// TwinCAT 3 PLC project PLC_ST40
// ProgramVersion: 3.1.4023.0
// libraries:
//   Tc2_DataExchange, * (Beckhoff Automation GmbH)
//   Tc2_IoFunctions, * (Beckhoff Automation GmbH)
//   Tc2_MC2, * (Beckhoff Automation GmbH)
//   Tc2_MC2_Drive, * (Beckhoff Automation GmbH)
//   Tc2_Standard, * (Beckhoff Automation GmbH)
//   Tc2_System, * (Beckhoff Automation GmbH)
//   Tc2_TcpIp, * (Beckhoff Automation GmbH)
//   Tc2_Utilities, * (Beckhoff Automation GmbH)
//   Tc3_EventLogger, * (Beckhoff Automation GmbH)
//   Tc3_Harman_MES_Interface, * (Harman)
//   Tc3_Module, * (Beckhoff Automation GmbH)
//   Tc3_Utilities_Extension, * (Harman)
// project tree:
//   DUTs/Camera/ ST_Camera_IN.TcDUT (not stored), ST_Camera_OUT.TcDUT (not stored)
//   DUTs/ENUMERATORs/ ENUM_AXIS_NAME.TcDUT, ENUM_CHANNEL.TcDUT, ENUM_PROCESS.TcDUT, ENUM_PROCESS_RESULT.TcDUT, ENUM_PROCESS_STATE.TcDUT, ENUM_SCREW_FEEDER.TcDUT, ENUM_SLOT.TcDUT, ENUM_SLOT_STATE.TcDUT, ENUM_SLOT_TYPE.TcDUT, ENUM_STATION.TcDUT
//   DUTs/ E_ADS_Cmd.TcTLEO (not stored), ST_CamSeq.TcDUT, ST_Coordinates_XYZ.TcDUT, ST_P1MesData.TcDUT, ST_PalletData.TcDUT, ST_PosData.TcDUT, ST_ProductData.TcDUT (not stored)
//   DUTs/Kuka/ ST_KRC_Control.TcDUT, ST_KRC_Status.TcDUT (not stored), U_KRC_Input.TcDUT, U_KRC_Output.TcDUT (not stored)
//   DUTs/NewFolder1/ ST_MOVE.TcDUT, ST_SCREWING.TcDUT, ST_SCR_RECIPE.TcDUT, ST_Vision.TcDUT
//   DUTs/PERSISTENT_STs/ ST_CONFIG.TcDUT
//   DUTs/STRUCTUREs/NewFolder1/ ST_MOVE_1.TcDUT, ST_SCREWING_1.TcDUT, ST_SCR_RECIPE_1.TcDUT
//   DUTs/STRUCTUREs/PROCESS_PARAM/MACHINE/ ST_P_BARCODE_READ.TcDUT, ST_P_CAMERA.TcDUT, ST_P_CHECK_INPUT.TcDUT, ST_P_MOVE.TcDUT, ST_P_RELEASE_PARTS.TcDUT, ST_P_RESET.TcDUT, ST_P_SCREWING.TcDUT, ST_P_SET.TcDUT, ST_P_SET_RECIPE.TcDUT, ST_P_SET_RECIPE_COND.TcDUT, ST_P_TAKE_SCREW.TcDUT, ST_P_WAIT.TcDUT, ST_P_WAIT_UNTIL.TcDUT
//   DUTs/STRUCTUREs/PROCESS_PARAM/MES/ ST_P_ASSY_ELEMENT.TcDUT, ST_P_CHECK_TIMECONTROL.TcDUT, ST_P_COMPLETE_ASSY.TcDUT, ST_P_COMPLETE_OP.TcDUT, ST_P_GET_CHILD.TcDUT, ST_P_GET_OP_STATE.TcDUT, ST_P_GET_PARENT.TcDUT, ST_P_GET_RECIPE.TcDUT, ST_P_RELEASE_MRT.TcDUT, ST_P_SAVE_MESDAT.TcDUT, ST_P_START_ASSY.TcDUT, ST_P_START_OP.TcDUT, ST_P_STOP_TIMECONTROL.TcDUT
//   DUTs/STRUCTUREs/ ST_COORDINATE.TcDUT, ST_DEPTH_DATA_DUT.TcDUT, ST_PARAMETER_COLLECTION.TcDUT, ST_PROCESS.TcDUT, ST_RECIPE.TcDUT, ST_SLOT_VISUALISATION.TcDUT
//   GVLs/ GVL_Constant.TcGVL, GVL_IO.TcGVL, GVL_Main.TcGVL, GVL_Persistenet.TcGVL, GVL_Recipe.TcGVL, GVL_Safety.TcGVL
//   / PlcTask.TcTTO
//   POUs/ Blink.TcPOU, Conveyor.TcPOU, Diag.TcPOU, Lift.TcPOU (not stored), MAIN.TcPOU, MesTest.TcPOU, P1_Camera.TcPOU, P2_Robot.TcPOU
//   POUs/FBs/ FB_ADSHandler.TcPOU (not stored), FB_BISL.TcPOU, FB_BISM.TcPOU, FB_Bistabil.TcPOU (not stored), FB_Conveyor.TcPOU, FB_Door.TcPOU, FB_FullCycleTime.TcPOU, FB_GenPulse.TcPOU (not stored), FB_KRC4.TcPOU, FB_Motor.TcPOU (not stored), FB_ReceipeList.TcPOU, FB_Stopper.TcPOU (not stored), FB_Stopper2.TcPOU (not stored), FB_TcEvent.TcPOU (not stored), FB_UpsC69xx.TcPOU, FB_UserLed.TcPOU, FB_WorkLight.TcPOU
//   POUs/FBs/FB_Camera/ FB_Kamino.TcPOU (not stored)
//   POUs/FBs/SmartLight/DUT/ E_BlinkFrequency.TcDUT (not stored), E_BuzzerType.TcDUT (not stored), E_Color.TcDUT, E_Mode.TcDUT (not stored)
//   POUs/FBs/SmartLight/ FB_SmartLight.TcPOU (not stored)
// real-time tasks:
//   TASK PlcTask: cycle T#10ms, priority 20, ADS port 350
// I/O:
//   DEVICE Device 4 (EtherCAT), AmsNetId 192.168.102.141.5.1
//     Term 1 (EK1100) [EK1100 EtherCAT Coupler (2A E-Bus)]
//       Term 2 (EL1918) [EL1918, 8Ch. Safety Input 24V, TwinSAFE]
//         modules: Module 2 (FSLOGIC)
//       Term 3 (EL2904) [EL2904, 4 Ch. Safety Output 24V, 0.5A, TwinSAFE]
//         modules: Module 1 (FSOES), Module 2 (DO)
//       Term 4 (EL2904) [EL2904, 4 Ch. Safety Output 24V, 0.5A, TwinSAFE]
//         modules: Module 1 (FSOES), Module 2 (DO)
//       Term 5 (EL1809) [EL1809 16Ch. Dig. Input 24V, 3ms]
//       Term 6 (EL1809) [EL1809 16Ch. Dig. Input 24V, 3ms]
//       Term 7 (EL1809) [EL1809 16Ch. Dig. Input 24V, 3ms]
//       Term 8 (EL6224) [EL6224 (IO Link Master)]
//       Term 9 (EL6224) [EL6224 (IO Link Master)]
//       Term 10 (EL9410) [EL9410 E-Bus Power Supplier  (Diagnostics)]
//       Term 11 (EL2809) [EL2809 16Ch. Dig. Output 24V, 0.5A]
//       Term 12 (EL2809) [EL2809 16Ch. Dig. Output 24V, 0.5A]
//       Term 13 (EL2809) [EL2809 16Ch. Dig. Output 24V, 0.5A]
//       Term 14 (EL2809) [EL2809 16Ch. Dig. Output 24V, 0.5A]
//       Term 17 (EL6070-0033) [EL6070-0033 1Ch. Licence key terminal, individual licences]
//       Term 36 (EL9011) [EL9011 End Terminal]
//     Drive 15 (AX5206-0000-0213) [AX5206-0000-0213 EtherCAT Drive (SoE, 2 Ch.)]
//       Term 16 (AX5805) [AX5805 (Safety Drive Option)]
//         modules: Module 1 (Safety Process Data, 2 axis), Module 2 (Standard Process Data, 2 axis)
//       Term 37 (EL9011) [EL9011 End Terminal]
//     KUKA (KRC4 secondary EL6695-1001) [KRC4 secondary EL6695-1001]
//       modules: Module 3 (Default IO)
//   DEVICE Device 1 (EtherCAT Automation Protocol), AmsNetId 192.168.102.141.2.1
//     Box 20 (ST10_TechEMYStopOn)
//     Box 21 (ST52_ConveyorReady)
//     Box 22 (ST40_TechEMYStopIgnored)
//     Box 24 (ST40_ConveyorReady)
//     Box 25 (ST40_Status)
// variable links:
//   Device 4 (EtherCAT) <-> Device 4 (EtherCAT)/Drive 15 (AX5206-0000-0213)/Term 16 (AX5805)
//     Term 1 (EK1100)/Term 2 (EL1918)/ConnectionOutputs/Message_8 RxPDO <-> Module 1 (Safety Process Data, 2 axis)/Inputs (Statusword)/FSOE
//   Device 4 (EtherCAT) <-> Device 4 (EtherCAT)/Term 1 (EK1100)/Term 2 (EL1918)
//     Drive 15 (AX5206-0000-0213)/Term 16 (AX5805)/Module 1 (Safety Process Data, 2 axis)/Outputs (Controlword)/FSOE <-> ConnectionInputs/Message_8 TxPDO
//     Term 1 (EK1100)/Term 3 (EL2904)/Module 1 (FSOES)/RxPDO/FSOE <-> ConnectionInputs/Message_7 TxPDO
//   Device 4 (EtherCAT) <-> Device 4 (EtherCAT)/Term 1 (EK1100)/Term 3 (EL2904)
//     Term 1 (EK1100)/Term 2 (EL1918)/ConnectionOutputs/Message_7 RxPDO <-> Module 1 (FSOES)/TxPDO/FSOE
//   PLC_ST40/PLC_ST40 Instance <-> Device 4 (EtherCAT)
//     PlcTask Inputs/Diag.FB_ECAT_DIAG.arrEcMasterNetId <-> InfoData/AmsNetId
//     PlcTask Inputs/Diag.FB_ECAT_DIAG.nEcMasterDevState <-> Inputs/DevState
//     PlcTask Inputs/Diag.FB_ECAT_DIAG.nEcMasterDeviceId <-> InfoData/DevId
//     PlcTask Inputs/Diag.FB_ECAT_DIAG.nEcMasterSlaveCount <-> Inputs/SlaveCount
//     PlcTask Inputs/Diag.FB_ECAT_DIAG.nEcMasterSlaveCountCfg <-> InfoData/CfgSlaveCount

CONFIGURATION PLC_ST40
    RESOURCE PLC ON TwinCAT3
        TASK PlcTask(INTERVAL := T#10ms, PRIORITY := 20);
        PROGRAM MAIN WITH PlcTask : MAIN;
    END_RESOURCE
END_CONFIGURATION

// ---- DUTs/ENUMERATORs/ENUM_AXIS_NAME.TcDUT
TYPE ENUM_AXIS_NAME :
(	
	CE_AXIS_X := 1,				// X-axis drive
	CE_AXIS_Y,					// Y-axis drive
	CE_AXIS_Z,					// Z-axis drive
	CE_AXIS_C, 					// C-axis drive
	CE_LAST_AXIS				(* placeholder, do not change*)
);
END_TYPE

// ---- DUTs/ENUMERATORs/ENUM_CHANNEL.TcDUT
TYPE ENUM_CHANNEL :
(
	Channel_1 := 0,
	Channel_2 := 1,
	Channel_3 := 2,
	Channel_4 := 3,
	Channel_5 := 4,
	Channel_6 := 5,
	Channel_7 := 6,
	Channel_8 := 7,
	Channel_9 := 8,
	Channel_10 := 9,
	Channel_11 := 10,
	Channel_12 := 11,
	Channel_13 := 12,
	Channel_14 := 13,
	Channel_15 := 14,
	Channel_16 := 15
);
END_TYPE

// ---- DUTs/ENUMERATORs/ENUM_PROCESS.TcDUT
TYPE ENUM_PROCESS :
(
	T_UNKNOWN:=0,

	//MACHINE
	T_MOVE:=1,
	T_TAKE_SCREW:=2,
	T_SCREWING:=3,
	T_BARCODE_READ:=4,
	T_CAMERA:=5,
	T_CHECK_INPUT:=6,
	T_WAIT:=7,
	T_WAIT_UNTIL:=8,
	T_SET:=9,
	T_RESET:=10,
	T_SET_RECIPE:=11,
	T_SET_RECIPE_COND:=12,
	T_RELEASE_PARTS:=13,
	
	//MES
	T_GET_OP_STATE:=14,
	T_GET_PARENT:=15,
	T_GET_CHILD:=16,
	T_START_OP:=17,
	T_SAVE_MESDAT:=18,
	T_COMPLETE_OP:=19,
	T_GET_RECIPE:=20,
	T_RELEASE_MRT:=21,
	T_START_ASSY:=22,
	T_ASSY_ELEMENT:=23,
	T_COMPLETE_ASSY:=24,
	T_CHECK_TIMECONTROL:=25,
	T_STOP_TIMECONTROL:=26,
	
	//LAST LINE INDICATOR
	T_END:=27
);
END_TYPE

// ---- DUTs/ENUMERATORs/ENUM_PROCESS_RESULT.TcDUT

TYPE ENUM_PROCESS_RESULT :
(
	FAILED := 0,
	PASSED := 1,
	CANCELD := 2,
	ABORTED := 3 
);
END_TYPE

// ---- DUTs/ENUMERATORs/ENUM_PROCESS_STATE.TcDUT
TYPE ENUM_PROCESS_STATE :
(
	TASK_READY:=0,
	TASK_BUSY,
	TASK_DONE,
	TASK_OK,
	TASK_NG
);
END_TYPE

// ---- DUTs/ENUMERATORs/ENUM_SCREW_FEEDER.TcDUT
TYPE ENUM_SCREW_FEEDER :
(
	CE_FEEDER_1 := 1,
	CE_FEEDER_2,
	CE_FEEDER_3,
	CE_FEEDER_4,
	CE_FEEDER_LAST
);
END_TYPE

// ---- DUTs/ENUMERATORs/ENUM_SLOT.TcDUT
TYPE ENUM_SLOT :
(
	SLOT_1 := 1,
	SLOT_2,
	SLOT_3,
	SLOT_4,
	SLOT_LAST
);
END_TYPE

// ---- DUTs/ENUMERATORs/ENUM_SLOT_STATE.TcDUT
TYPE ENUM_SLOT_STATE :
(
	EMPTY := 0,
	IN_QUEUE,
	WAIT_FOR_START,
	DISABLED,
	IN_WORK,
	FINISHED
);
END_TYPE

// ---- DUTs/ENUMERATORs/ENUM_SLOT_TYPE.TcDUT
TYPE ENUM_SLOT_TYPE :
(
	SETUP := 0,
	LOGIC := 1,
	TEARDOWN := 2
);
END_TYPE

// ---- DUTs/ENUMERATORs/ENUM_STATION.TcDUT
{attribute 'strict'}
{attribute 'to_string'}
TYPE ENUM_STATION :
(
	SCREWING:= 0,
	GSL:= 1,
	DISPENSER:= 2
);
END_TYPE

// ---- DUTs/Kuka/ST_KRC_Control.TcDUT
TYPE ST_KRC_Control :
STRUCT
(*-----=== Byte 00 ===-----*)
	bPgnoParity				:BIT;				// 00.0	Parity BIT FOR PROGRAM number check (NOT used)
	bPgnoValid				:BIT;				// 00.1	Program number is read for this signal's rising edge
	bExtStart				:BIT;				// 00.2	Start cell.src program (not used)
	bMoveEnable				:BIT;				// 00.3	Enable signal for movement
	bConfMess				:BIT;				// 00.4	Message confirmation message
	bDrivesOff				:BIT;				// 00.5	Turn off drives if this signal is FALSE at least for 20 ms (nem használt)
	bDrivesOn				:BIT;				// 00.6	Turn on drives if this signal is TRUE at least for 20 ms
	bIOAct					:BIT;				// 00.7	Enable external control (not used)

(*-----=== Byte 01 ===-----*)
	{attribute 'hide'}
	_reserved_01			:BYTE;				// 01	Tartalék	

(*-----=== Byte 02 ===-----*)
	nProgNr					:BYTE;				// 02	Program number
	
(*-----=== Byte 03 ===-----*)
	{attribute 'hide'}
	_reserved_03			:BYTE;				// 03	Tartalék (Safety IO)	

(*-----=== Byte 04 ===-----*)
	bEnableMoveInPalettZone	:BIT;				// 04.0	Enabling Robot to move insdie Palett Zone after it requested it
	{attribute 'hide'}
	_reserved_04_1			:BIT;				// 04.1	Tartalék	
	{attribute 'hide'}
	_reserved_04_2			:BIT;				// 04.2	Tartalék	
	{attribute 'hide'}
	_reserved_04_3			:BIT;				// 04.3	Tartalék	
	{attribute 'hide'}
	_reserved_04_4			:BIT;				// 04.4	Tartalék	
	{attribute 'hide'}
	_reserved_04_5			:BIT;				// 04.5	Tartalék	
	{attribute 'hide'}
	_reserved_04_6			:BIT;				// 04.6	Tartalék	
	{attribute 'hide'}
	_reserved_04_7			:BIT;				// 04.7	Tartalék	
	
(*-----=== Byte 05 ===-----*)
	bVacuumErrorClear		:BIT;				// 05.0	Clearing Vacuum Error
	{attribute 'hide'}
	_reserved_05_1			:BIT;				// 05.1	Tartalék	
	{attribute 'hide'}
	_reserved_05_2			:BIT;				// 05.2	Tartalék	
	{attribute 'hide'}
	_reserved_05_3			:BIT;				// 05.3	Tartalék	
	{attribute 'hide'}
	_reserved_05_4			:BIT;				// 05.4	Tartalék	
	{attribute 'hide'}
	_reserved_05_5			:BIT;				// 05.5	Tartalék	
	{attribute 'hide'}
	_reserved_05_6			:BIT;				// 05.6	Tartalék	
	{attribute 'hide'}
	_reserved_05_7			:BIT;				// 05.7	Tartalék	
	
(*-----=== Byte 06 ===-----*)
	{attribute 'hide'}
	_reserved_06			:BYTE;				// 06	Tartalék	
(*-----=== Byte 07 ===-----*)
	{attribute 'hide'}
	_reserved_07			:BYTE;				// 07	Tartalék	
(*-----=== Byte 08 ===-----*)
	{attribute 'hide'}
	_reserved_08			:BYTE;				// 08	Tartalék	
(*-----=== Byte 09 ===-----*)
	{attribute 'hide'}
	_reserved_09			:BYTE;				// 09	Tartalék
(*-----=== Byte 10 ===-----*)
	{attribute 'hide'}
	_reserved_10			:BYTE;				// 10	Tartalék
(*-----=== Byte 11 ===-----*)
	{attribute 'hide'}
	_reserved_11			:BYTE;				// 11	Tartalék
(*-----=== Byte 12 ===-----*)
	{attribute 'hide'}
	_reserved_12			:BYTE;				// 12	Tartalék
(*-----=== Byte 13 ===-----*)
	{attribute 'hide'}
	_reserved_13			:BYTE;				// 13	Tartalék	
(*-----=== Byte 14 ===-----*)
	{attribute 'hide'}
	_reserved_14			:BYTE;				// 14	Tartalék	
(*-----=== Byte 15 ===-----*)
	{attribute 'hide'}
	_reserved_15			:BYTE;				// 15	Tartalék	
END_STRUCT
END_TYPE

// ---- DUTs/Kuka/U_KRC_Input.TcDUT
TYPE U_KRC_Input :
UNION
	aStdIn		AT %I*		:ARRAY [0..3] OF DWORD;
	Status					:ST_KRC_Status;	
END_UNION
END_TYPE

// ---- DUTs/NewFolder1/ST_MOVE.TcDUT
TYPE ST_MOVE :
STRUCT
	Target:					ST_COORDINATE;
	Override:				LREAL;
	Comment:				STRING(255);
END_STRUCT
END_TYPE

// ---- DUTs/NewFolder1/ST_SCREWING.TcDUT
TYPE ST_SCREWING :
STRUCT
	Target:					ST_COORDINATE;
	Override:				LREAL;
	Feeder:					ENUM_SCREW_FEEDER;
	Comment:				STRING(255);
	PositionNumber:			INT;
	ScrewingProgramId:		INT;
	PreScrewingOn:			BOOL;
	PreScrewingProgramId:	INT;
	LastPosition:			BOOL:=TRUE;
END_STRUCT
END_TYPE

// ---- DUTs/NewFolder1/ST_SCR_RECIPE.TcDUT
TYPE ST_SCR_RECIPE :
	STRUCT
		Descr:				STRING(MAX_STRING_LENGTH);
		Name:				STRING(MAX_STRING_LENGTH);
		Seq:				ARRAY[0..99] OF ST_Vision;
	END_STRUCT
END_TYPE

// ---- DUTs/NewFolder1/ST_Vision.TcDUT
TYPE ST_Vision :
STRUCT
	Target:					ST_COORDINATE;
	Comment:				STRING(255);
	PositionNumber:			INT;
	CheckingProgramId:		INT;
	LastPosition:			BOOL:=TRUE;
END_STRUCT
END_TYPE

// ---- DUTs/PERSISTENT_STs/ST_CONFIG.TcDUT
TYPE ST_CONFIG :
STRUCT
	AXIS_POSITION_TOLERANCE:		LREAL;
	AXIS_OVERRIDE:					LREAL;
	AXIS_C_EXIST:					BOOL;	
	AXIS_END_SENSOR_EXIST:			BOOL;
	STATION_ID:						INT;
	ADAPTER_ID:						UINT;
	NUMBER_OF_SLOTS:				INT:=4;
	CUSTOM_POSITIONS:				ARRAY[0..19] OF ST_MOVE;
	//Depth measurement check ON/OFF	
	DEPTH_MEASURE_ON:				BOOL:=TRUE;	
	DEPTH_TRIGGER_OFFSET :			LREAL;
	DEPTH_TOLERANCE :				LREAL;
	//Screw length check ON/OFF
	SCREW_CHECK_ON:					BOOL:=TRUE;
	SCREW_LENGTH:					ARRAY [CE_FEEDER_1..(CE_FEEDER_LAST-1)] OF LREAL;
	SCREW_LENGTH_TOLERANCE:			LREAL;		
	//X axis specific positions:
	POS_X_CHANGE_WP:				LREAL;
	POS_X_HOME:						LREAL;
	POS_X_SAFETY:					LREAL;	
	//Y axis specific positions:
	POS_Y_SCREW_FEEDER:				ARRAY [CE_FEEDER_1..(CE_FEEDER_LAST-1)] OF LREAL;
	POS_Y_SCREW_DROP:				ARRAY [CE_FEEDER_1..(CE_FEEDER_LAST-1)] OF LREAL;	
	//Z axis specific positions:
	POS_Z_SCREW_FEEDER:				ARRAY [CE_FEEDER_1..(CE_FEEDER_LAST-1)] OF LREAL;
	POS_Z_SCREW_DROP:				ARRAY [CE_FEEDER_1..(CE_FEEDER_LAST-1)] OF LREAL;
	POS_Z_HOME:						LREAL;
	POS_Z_SAFETY:					LREAL;	
	//C axis specific positions:
	POS_C_HOME:						LREAL;
	
	(* Configuration variables for GSL Application *)	
	(* Configuration variables for Dispensing Application *)
END_STRUCT
END_TYPE

// ---- DUTs/STRUCTUREs/NewFolder1/ST_MOVE_1.TcDUT
TYPE ST_MOVE_1 :
STRUCT
	Target:					ST_COORDINATE;
	Override:				LREAL;
	Comment:				STRING(255);
END_STRUCT
END_TYPE

// ---- DUTs/STRUCTUREs/NewFolder1/ST_SCREWING_1.TcDUT
TYPE ST_SCREWING_1 :
STRUCT
	Target:					ST_COORDINATE;
	Override:				LREAL;
	Feeder:					ENUM_SCREW_FEEDER;
	Comment:				STRING(255);
	PositionNumber:			INT;
	ScrewingProgramId:		INT;
	PreScrewingOn:			BOOL;
	PreScrewingProgramId:	INT;
	LastPosition:			BOOL:=TRUE;
END_STRUCT
END_TYPE

// ---- DUTs/STRUCTUREs/NewFolder1/ST_SCR_RECIPE_1.TcDUT
TYPE ST_SCR_RECIPE_1 :
	STRUCT
		Descr:				STRING(MAX_STRING_LENGTH);
		Name:				STRING(MAX_STRING_LENGTH);
		Seq:				ARRAY[0..99] OF ST_SCREWING;
	END_STRUCT
END_TYPE

// ---- DUTs/STRUCTUREs/PROCESS_PARAM/MACHINE/ST_P_BARCODE_READ.TcDUT
TYPE ST_P_BARCODE_READ :
STRUCT
	IpAddress:					STRING;
	Port:						STRING;
	Start:						STRING;
	End:						STRING;
	Error:						STRING;
	Barcode:					INT;
END_STRUCT
END_TYPE

// ---- DUTs/STRUCTUREs/PROCESS_PARAM/MACHINE/ST_P_CAMERA.TcDUT
TYPE ST_P_CAMERA :
STRUCT
	ProgramName:			STRING;
END_STRUCT
END_TYPE

// ---- DUTs/STRUCTUREs/PROCESS_PARAM/MACHINE/ST_P_CHECK_INPUT.TcDUT
TYPE ST_P_CHECK_INPUT :
STRUCT
	Block:		INT;
	Channel:	ENUM_CHANNEL;
	State:		BOOL;
END_STRUCT
END_TYPE

// ---- DUTs/STRUCTUREs/PROCESS_PARAM/MACHINE/ST_P_MOVE.TcDUT
TYPE ST_P_MOVE :
STRUCT
	Override:			LREAL;
	X:					LREAL;
	Y:					LREAL;
	Z:					LREAL;
	C:					LREAL;
END_STRUCT
END_TYPE

// ---- DUTs/STRUCTUREs/PROCESS_PARAM/MACHINE/ST_P_RELEASE_PARTS.TcDUT
TYPE ST_P_RELEASE_PARTS :
STRUCT
	Override:		LREAL;
	Feeder:			ENUM_SCREW_FEEDER;
END_STRUCT
END_TYPE

// ---- DUTs/STRUCTUREs/PROCESS_PARAM/MACHINE/ST_P_RESET.TcDUT
TYPE ST_P_RESET :
STRUCT
	Block:		INT;
	Channel:	ENUM_CHANNEL;
	ExecuteOnFail:	BOOL;
END_STRUCT
END_TYPE

// ---- DUTs/STRUCTUREs/PROCESS_PARAM/MACHINE/ST_P_SCREWING.TcDUT
TYPE ST_P_SCREWING :
STRUCT
	PreScrewingActive:				BOOL;
	PreScrewingPrg:					INT;
	ScrewingPrg:					INT;
	PosNumber:						INT;
END_STRUCT
END_TYPE

// ---- DUTs/STRUCTUREs/PROCESS_PARAM/MACHINE/ST_P_SET.TcDUT
TYPE ST_P_SET :
STRUCT
	Block:		INT;
	Channel:	ENUM_CHANNEL;
	ExecuteOnFail:	BOOL;
END_STRUCT
END_TYPE

// ---- DUTs/STRUCTUREs/PROCESS_PARAM/MACHINE/ST_P_SET_RECIPE.TcDUT
TYPE ST_P_SET_RECIPE :
STRUCT
	RecipeName:			STRING;
END_STRUCT
END_TYPE

// ---- DUTs/STRUCTUREs/PROCESS_PARAM/MACHINE/ST_P_SET_RECIPE_COND.TcDUT
TYPE ST_P_SET_RECIPE_COND :
STRUCT
	RecipeName:					STRING;
END_STRUCT
END_TYPE

// ---- DUTs/STRUCTUREs/PROCESS_PARAM/MACHINE/ST_P_TAKE_SCREW.TcDUT
TYPE ST_P_TAKE_SCREW :
STRUCT
	//'X:=-86.36;Y:=168.56;Z:=115.23;C:=90.12;FEEDER:=2;'
	Feeder:				INT;
	Override:			LREAL;
	X:					LREAL;
	Y:					LREAL;
	Z:					LREAL;
	C:					LREAL;
END_STRUCT
END_TYPE

// ---- DUTs/STRUCTUREs/PROCESS_PARAM/MACHINE/ST_P_WAIT.TcDUT
TYPE ST_P_WAIT :
STRUCT
	WaitTime:		INT;
	ExecuteOnFail:	BOOL;
END_STRUCT
END_TYPE

// ---- DUTs/STRUCTUREs/PROCESS_PARAM/MACHINE/ST_P_WAIT_UNTIL.TcDUT
TYPE ST_P_WAIT_UNTIL :
STRUCT
	Block:		INT;
	Channel:	ENUM_CHANNEL;
	State:		BOOL;
	ExecuteOnFail:	BOOL;
END_STRUCT
END_TYPE

// ---- DUTs/STRUCTUREs/PROCESS_PARAM/MES/ST_P_ASSY_ELEMENT.TcDUT
TYPE ST_P_ASSY_ELEMENT :
STRUCT
	LeadingSFC:				INT;
	InventoriID:			INT;
END_STRUCT
END_TYPE

// ---- DUTs/STRUCTUREs/PROCESS_PARAM/MES/ST_P_CHECK_TIMECONTROL.TcDUT
TYPE ST_P_CHECK_TIMECONTROL :
STRUCT
	Barcode:			INT;
	ControlName:		STRING;
END_STRUCT
END_TYPE

// ---- DUTs/STRUCTUREs/PROCESS_PARAM/MES/ST_P_COMPLETE_ASSY.TcDUT
TYPE ST_P_COMPLETE_ASSY :
STRUCT
END_STRUCT
END_TYPE

// ---- DUTs/STRUCTUREs/PROCESS_PARAM/MES/ST_P_COMPLETE_OP.TcDUT
TYPE ST_P_COMPLETE_OP :
STRUCT
	SetIndex:				BOOL;
	Index:					INT;
	Barcode:			INT;
END_STRUCT
END_TYPE

// ---- DUTs/STRUCTUREs/PROCESS_PARAM/MES/ST_P_GET_CHILD.TcDUT
TYPE ST_P_GET_CHILD :
STRUCT
	Position:				INT;
	ContainerId:			INT;
	Barcode:				INT;
END_STRUCT
END_TYPE

// ---- DUTs/STRUCTUREs/PROCESS_PARAM/MES/ST_P_GET_OP_STATE.TcDUT
TYPE ST_P_GET_OP_STATE :
STRUCT
	CheckState:				BOOL;
	OperationName:			STRING;
	OperationIndex:			INT;
	Barcode:				INT;
END_STRUCT
END_TYPE

// ---- DUTs/STRUCTUREs/PROCESS_PARAM/MES/ST_P_GET_PARENT.TcDUT
TYPE ST_P_GET_PARENT :
STRUCT
	ContainerId:			INT;
	Barcode:				INT;
END_STRUCT
END_TYPE

// ---- DUTs/STRUCTUREs/PROCESS_PARAM/MES/ST_P_GET_RECIPE.TcDUT
TYPE ST_P_GET_RECIPE :
STRUCT
	Barcode:				INT;
	ByCustomField:			BOOL;
	CustomFiled:			STRING;
	Contains:				STRING;
END_STRUCT
END_TYPE

// ---- DUTs/STRUCTUREs/PROCESS_PARAM/MES/ST_P_RELEASE_MRT.TcDUT
TYPE ST_P_RELEASE_MRT :
STRUCT
END_STRUCT
END_TYPE

// ---- DUTs/STRUCTUREs/PROCESS_PARAM/MES/ST_P_SAVE_MESDAT.TcDUT
TYPE ST_P_SAVE_MESDAT :
STRUCT
	SetIndex:				BOOL;
	Index:					INT;
	Barcode:				INT;
END_STRUCT
END_TYPE

// ---- DUTs/STRUCTUREs/PROCESS_PARAM/MES/ST_P_START_ASSY.TcDUT
TYPE ST_P_START_ASSY :
STRUCT
	Barcode:				INT;
END_STRUCT
END_TYPE

// ---- DUTs/STRUCTUREs/PROCESS_PARAM/MES/ST_P_START_OP.TcDUT
TYPE ST_P_START_OP :
STRUCT
	SetIndex:				BOOl;
	Index:					INT;
	Barcode:				INT;
END_STRUCT
END_TYPE

// ---- DUTs/STRUCTUREs/PROCESS_PARAM/MES/ST_P_STOP_TIMECONTROL.TcDUT
TYPE ST_P_STOP_TIMECONTROL :
STRUCT
	Barcode:			INT;
	ControlName:		STRING;
END_STRUCT
END_TYPE

// ---- DUTs/STRUCTUREs/ST_COORDINATE.TcDUT
TYPE ST_COORDINATE :
STRUCT
	X: LREAL;
	Y: LREAL;
	Z: LREAL;
	C: LREAL;
END_STRUCT
END_TYPE

// ---- DUTs/STRUCTUREs/ST_DEPTH_DATA_DUT.TcDUT
TYPE ST_DEPTH_DATA_DUT :
STRUCT
	lrDepth_MV:			LREAL;
	lrDepth_LL:			LREAL;
	lrDepth_UL:			LREAL;
	lrDepth_Signal:		LREAL;
END_STRUCT
END_TYPE

// ---- DUTs/STRUCTUREs/ST_PARAMETER_COLLECTION.TcDUT
TYPE ST_PARAMETER_COLLECTION :
STRUCT
	//MACHINE
	ST_P_MOVE:				ST_P_MOVE;
	ST_P_TAKE_SCREW:		ST_P_TAKE_SCREW;
	ST_P_SCREWING:			ST_P_SCREWING;
	ST_P_BARCODE_READ:		ST_P_BARCODE_READ;
	ST_P_CAMERA:			ST_P_CAMERA;
	ST_P_CHECK_INPUT:		ST_P_CHECK_INPUT;
	ST_P_WAIT:				ST_P_WAIT;
	ST_P_WAIT_UNTIL:		ST_P_WAIT_UNTIL;
	ST_P_SET:				ST_P_SET;
	ST_P_RESET:				ST_P_RESET;
	ST_P_SET_RECIPE:		ST_P_SET_RECIPE;
	ST_P_SET_RECIPE_COND:	ST_P_SET_RECIPE_COND;
	ST_P_RELEASE_PARTS:		ST_P_RELEASE_PARTS;
	
	//MES
	ST_P_GET_OP_STATE:		ST_P_GET_OP_STATE;
	ST_P_GET_PARENT:		ST_P_GET_PARENT;
	ST_P_GET_CHILD:			ST_P_GET_CHILD;
	ST_P_START_OP:			ST_P_START_OP;
	ST_P_SAVE_MESDAT:		ST_P_SAVE_MESDAT;
	ST_P_COMPLETE_OP:		ST_P_COMPLETE_OP;
	ST_P_GET_RECIPE:		ST_P_GET_RECIPE;
	ST_P_RELEASE_MRT:		ST_P_RELEASE_MRT;
	ST_P_START_ASSY:		ST_P_START_ASSY;
	ST_P_ASSY_ELEMENT:		ST_P_ASSY_ELEMENT;
	ST_P_COMPLETE_ASSY:		ST_P_COMPLETE_ASSY;
	ST_P_CHECK_TIMECONTROL:	ST_P_CHECK_TIMECONTROL;
	ST_P_STOP_TIMECONTROL:	ST_P_STOP_TIMECONTROL;
END_STRUCT
END_TYPE

// ---- DUTs/STRUCTUREs/ST_PROCESS.TcDUT
TYPE ST_PROCESS :
STRUCT
	ChageSlot:			BOOL:=FALSE;	(* Change slot after finished this position TASK *)	
	ProcessType:		ENUM_PROCESS;		(* Describe what we want to do in *)
	Comment:			STRING(255);
	Parameter:			STRING(255);
END_STRUCT
END_TYPE

// ---- DUTs/STRUCTUREs/ST_RECIPE.TcDUT
TYPE ST_RECIPE :
STRUCT	
	DESCRIPTION:		STRING(MAX_STRING_LENGTH);
	NAME:				STRING(MAX_STRING_LENGTH);
	PROCESS_LIST:		ARRAY [0..299] OF STRING(MAX_STRING_LENGTH);	
END_STRUCT
END_TYPE

// ---- DUTs/STRUCTUREs/ST_SLOT_VISUALISATION.TcDUT
TYPE ST_SLOT_VISUALISATION :
STRUCT
	CurrentStep:		STRING(255);
	Comment:			STRING(255);
	State:				INT;
	Progress:			LREAL;
END_STRUCT
END_TYPE

// ---- DUTs/ST_CamSeq.TcDUT
TYPE ST_CamSeq :
STRUCT
	rAxisX			:REAL;
	rAxisY			:REAL;
	nCamProg		:UINT;
	bExecute		:BOOL;
END_STRUCT
END_TYPE

// ---- DUTs/ST_Coordinates_XYZ.TcDUT
TYPE ST_Coordinates_XYZ :
STRUCT
	PosX: REAL;
	PosY: REAL;
	PosZ: REAL;
END_STRUCT
END_TYPE

// ---- DUTs/ST_P1MesData.TcDUT
TYPE ST_P1MesData :
STRUCT
	sDMC_Code			:STRING;
	nOP_Index			:INT;
	sOP_Name			:STRING;
	sOP_CustomData		:STRING(1000);
	sOP_ReceipeList		:STRING(1000);
END_STRUCT
END_TYPE

// ---- DUTs/ST_PalletData.TcDUT
TYPE ST_PalletData :
STRUCT
		sCarrierCode		:STRING(40);
		sCoverCode 			:STRING(40);
		sPCBACode			:STRING(40);
		sFanCode			:STRING(40);
		sMRTCode			:STRING(40);
		nPalletState 		:WORD;		// Paletta státus:	0	Üres paletta
										//					1	Selejt
										//					2	OK termék a palettán
										//					10	ST10 Teszt paletta
										//					11	ST11 Teszt paletta
										//					20	ST20 Teszt paletta
										//					30	ST30 Teszt paletta
										//					41	ST40 Kamera Teszt paletta
										//					42	ST40 Robot Teszt paletta
										//					51	ST51 Teszt paletta
										//					51	ST52 Teszt paletta
										//					70	ST70 Teszt paletta
										//					60	ST60 Teszt paletta
		nPalletCommand		:WORD;		//	Teszt paletta parancs

		nDone				:WORD;		//Állomás kész bitek
										//nDone.0		ST10		Operátor pozíció
										//nDone.1		ST11		Nyomtató
										//nDone.2		ST20		Diszpenzáló I.
										//nDone.3		ST30		Diszpenzáló II.		-majd ha egyszer lesz
										//nDone.4		ST40.1		Kamerás ell.		
										//nDone.5		ST40.2		Robot
										//nDone.6		ST50/1		Csavarozó I. 		-majd ha egyszer lesz
										//nDone.7		ST50/2		Csavarozó II.
										//nDone.8		ST70		Jótermék kirakó
										//nDone.9		ST60		Selejt kirakó
		nErrorCode			:WORD;
		stInventoryList		:ST_INVENTORY_LIST;
END_STRUCT
END_TYPE

// ---- DUTs/ST_PosData.TcDUT
TYPE ST_PosData :
STRUCT
	nState				:UDINT;
	nStateLast			:UDINT;
	sState				:STRING;
	bBusy				:BOOL;
	bReady				:BOOL;
	bPass				:BOOL;
	bFail				:BOOL;
	bError				:BOOL;
	nErrorCode			:UDINT;
	nCycleTime			:REAL;
	bManualModeEnable	:BOOL;
	bDoorOpenEnable		:BOOL;
	stProductData		:ST_ProductData;
END_STRUCT
END_TYPE

// ---- POUs/FBs/SmartLight/DUT/E_Color.TcDUT
{attribute 'qualified_only'}
{attribute 'strict'}
TYPE E_Color :
(
	off,green,red,yellow,blue,orange
);
END_TYPE

// ---- GVLs/GVL_Constant.TcGVL
VAR_GLOBAL CONSTANT
	nP1CheckSim_Index					:INT := 0;					// Sim kártya ellenőrzés
	nP1CheckComponent_Index				:INT := 1;					// Ventilátor ellenőrzés
	nP2Assy_Auto2_Index					:INT := 2;					// Összeszerelés	
	nP1GapFillerCheckCover_Index		:INT := 3;					// "Gapfiller" ellenőrzés
	nP1SupplierInport_Index				:INT := 4;					// Örökbe fogadás majd ha kell pl.: a ventilátorhoz

	nNbrOfAlarms						:UINT := 13;	

	
(*
Inventory sorrend
0:	MRT
1:	Carrier
2:	Cover
3:	PCBA
4:	Fan
*)


END_VAR

// ---- GVLs/GVL_IO.TcGVL
VAR_GLOBAL
	(* Digital input A1*)
	i_bLop1				AT %I*		:BOOL;			// I2.1
	i_bLop2				AT %I*		:BOOL;			// I2.2
													// I2.3			Tartalék
	i_bAirOK			AT %I*		:BOOL;			// I2.4
	i_bDoorOpenBtn		AT %I*		:BOOL;			// I2.5
													// I2.6			Tartalék
	i_bDC1OK			AT %I*		:BOOL;			// I2.7
	i_bDC2OK			AT %I*		:BOOL;			// I2.8
	
//	i_bConvejor1OK		AT %I*		:BOOL;			// I2.9			FB-hez linkelve
//	i_bConvejor2OK		AT %I*		:BOOL;			// I2.10		FB-hez linkelve
//	i_bConvejor3OK		AT %I*		:BOOL;			// I2.11		FB-hez linkelve
//	i_bConvejor4OK		AT %I*		:BOOL;			// I2.12		FB-hez linkelve
//	i_bConvejor5OK		AT %I*		:BOOL;			// I2.13		FB-hez linkelve
//	i_bConvejor6OK		AT %I*		:BOOL;			// I2.14		Tartalék
													// I2.15		Tartalék
													// I2.16		Tartalék
	
													// I3.1			Tartalék
													// ...			Tartalék
													// I3.16		Tartalék

	(* Digital input A6*)		//LI+1
	q_bGreenBtnLed		AT %Q*		:BOOL;			// Q11.1
	q_bRedBtnLed		AT %Q*		:BOOL;			// Q11.2
	q_bWhiteBtnLed		AT %Q*		:BOOL;			// Q11.3
													// Q11.4		Tartalék
													// ...			Tartalék
													// Q11.8		Tartalék
	q_bAreaLighting		AT %Q*		:BOOL;			// Q11.9
	q_bLockDoor			AT %Q*		:BOOL;			// Q11.10
													// Q11.11		Tartalék
													// ...			Tartalék
													// Q11.16		Tartalék

	(* Digital input A7*)		//LI+1
													// Q12.1		Tartalék
													// ...			Tartalék
													// Q12.16		Tartalék
	
	(* Digital input A9*)		//LO+1
//	q_bConvejor1On		AT %Q*		:BOOL;			// Q21.1		FB-hez linkelve
//	q_bConvejor2On		AT %Q*		:BOOL;			// Q21.2		FB-hez linkelve
//	q_bConvejor3On		AT %Q*		:BOOL;			// Q21.3		FB-hez linkelve
//	q_bConvejor4On		AT %Q*		:BOOL;			// Q21.4		FB-hez linkelve
//	q_bConvejor5On		AT %Q*		:BOOL;			// Q21.5		FB-hez linkelve
//	q_bConvejor6On		AT %Q*		:BOOL;			// Q21.6		Tartalék
//	q_bStopper1			AT %Q*		:BOOL;			// Q21.7		FB-hez linkelve
//	q_bStopper2			AT %Q*		:BOOL;			// Q21.8		FB-hez linkelve

//	q_bStopper3			AT %Q*		:BOOL;			// Q21.9		FB-hez linkelve
//	q_bStopper4			AT %Q*		:BOOL;			// Q21.10		FB-hez linkelve
//	q_bStopper5			AT %Q*		:BOOL;			// Q21.11		FB-hez linkelve
//	q_bStopper6			AT %Q*		:BOOL;			// Q21.12		FB-hez linkelve
													// Q21.13		Tartalék
													// ...			Tartalék
													// Q11.16		Tartalék
													
	(* Digital input A11*)		//LO+2
//	q_bP1LiftWorkPos	AT %Q*		:BOOL;			// Q31.1		FB-hez linkelve
//	q_bP1LiftBasePos	AT %Q*		:BOOL;			// Q31.2		FB-hez linkelve
//	q_bP2LiftWorkPos	AT %Q*		:BOOL;			// Q31.3		FB-hez linkelve
//	q_bP2LiftBasePos	AT %Q*		:BOOL;			// Q31.4		FB-hez linkelve
													// Q31.5		Tartalék
													// ...			Tartalék
													// Q11.16		Tartalék
													
	(* IOLink A3*)
	(*IOL1*)
//	i_bStopperSensor1	AT %I*		:BOOL;			// IOL 1.0.4	FB-hez linkelve
//	i_bStopperSensor2	AT %I*		:BOOL;			// IOL 1.1.4	FB-hez linkelve
//	i_bStopperSensor3	AT %I*		:BOOL;			// IOL 1.2.4	FB-hez linkelve
//	i_bP1LiftWorkPos	AT %I*		:BOOL;			// IOL 1.3.4	FB-hez linkelve
	i_bP2PalletSensor	AT %I*		:BOOL;			// IOL 1.4.4	P1 és P2 közötti nemkívánatos paletta érzékelése
													// IOL 1.5.4	Tartalék
													// ...			Tartalék
													// IOL 1.7.4	Tartalék

													// IOL 1.0.2	Tartalék
													// IOL 1.1.2	Tartalék
													// IOL 1.2.2	Tartalék
//	i_bP1LiftBasePos	AT %I*		:BOOL;			// IOL 1.3.2	FB-hez linkelve
													// IOL 1.4.2	Tartalék
													// ...			Tartalék
													// IOL 1.7.2	Tartalék
													
	(*IOL2*)
//	i_bStopperSensor4	AT %I*		:BOOL;			// IOL 2.0.4	FB-hez linkelve
//	i_bStopperSensor5	AT %I*		:BOOL;			// IOL 2.1.4	FB-hez linkelve
//	i_bStopperSensor6	AT %I*		:BOOL;			// IOL 2.2.4	FB-hez linkelve
//	i_bP2LiftWorkPos	AT %I*		:BOOL;			// IOL 2.3.4	FB-hez linkelve
	i_bP2DutSensor1		AT %I*		:BOOL;			// IOL 2.4.4	PCB
	i_bP2DutSensor2		AT %I*		:BOOL;			// IOL 2.5.4	Cover
	i_bP2DutSensor3		AT %I*		:BOOL;			// IOL 2.6.4	Carrier
	i_bP2DutSensor4		AT %I*		:BOOL;			// IOL 2.7.4	FAN

													// IOL 2.0.2	Tartalék
													// IOL 2.1.2	Tartalék
													// IOL 2.2.2	Tartalék
//	i_bP2LiftBasePos	AT %I*		:BOOL;			// IOL 2.3.2	FB-hez linkelve
													// IOL 2.4.2	Tartalék
													// ...			Tartalék
													// IOL 2.7.2	Tartalék

	(*IOL3*)
													//				Tartalék
	(*IOL4*)
													//				Tartalék

	(* IOLink A4*)
	(*IOL5*)
//	BNI IOL-801-102-Z037							//	Toronylámpa
	(*IOL6*)
//	BIS014K											//	P1 RFID olvaasó
	(*IOL7*)
//	BIS014K											//	P2 RFID olvaasó
	(*IOL8*)
													//				Tartalék
													
	(* EAP Var *)
	i_bST10_TechEMYStopOn				AT %I*		:BOOL;
	i_bST10_TechEMYStopOn_Quality		AT %I*		:UINT;

	i_bST51_ConveyorReady				AT %I*		:BOOL;			
	i_nST51_ConveyorReady_Quality		AT %I*		:UINT;
	
	q_bST40_ConveyorReady				AT %Q*		:BOOL;			
	q_bST40_TechEMYStopIgnored			AT %Q*		:BOOL;

	q_bST40_Status						AT %Q*		:DWORD;		//	.00			Processz státusz
																//	.01
																//	.02
																//	.03
																//	.04
																//	.05
																//	.06
																//	.07
																//	.08			Hiba
																//	.09			Anyagkifogyás
																//	.10
																//	.11
																//	.12
																//	.13
																//	.14
																//	.15
																//	.16
																//	.17
																//	.18
																//	.19
																//	.20
																//	.21
																//	.22
																//	.23
																//	.24
																//	.25
																//	.26
																//	.27
																//	.28
																//	.29
																//	.30
																//	.31		
END_VAR

// ---- GVLs/GVL_Main.TcGVL
VAR_GLOBAL
(* Blink *)
	bBL50p50						:BOOL;				(*50ms/50ms*)
	bBL100p100						:BOOL;				(*100ms/100ms*)
	bBL250p250						:BOOL;				(*250ms/250ms*)
	bBL500p500						:BOOL;				(*500ms/500ms*)
	bBL1000p1000					:BOOL;				(*1000ms/1000ms*)
	bBL250p750						:BOOL;				(*750ms/250ms*)
	bTakt100ms						:BOOL;				(*Takt 100ms*)
	bTakt200ms						:BOOL;				(*Takt 200ms*)
	bTakt500ms						:BOOL;				(*Takt 500ms*)
	bTakt1s							:BOOL;				(*Takt 1000ms*)
	bTakt2s							:BOOL;				(*Takt 2000ms*)
	nLifeSignal						:UINT;

(* Main *)
	bManualMode						:BOOL;				(* Kézi üzemmód gépállapot *)
	bManualModeRequest				:BOOL;
	sMode							:STRING;			(* Aktuális üzemmód *)
	nMode							:BYTE;
	nLocale							:BYTE;
	bEcoMode						:BOOL;				(* Eco mód *)
	rtStep							:R_Trig;			(* Léptetés trigger*)
	bStepMode						:BOOL;				(* Léptetés mód *)
	bStepP							:BOOL;				(* Léptetés impulzus *)
	bStepHMI						:BOOL;				(* Léptetés gomb HMI *)
	bStepEnable						:BOOL;				(* Léphet a folyamat*)
	bAckHMI							:BOOL;				(* Nyugta HMI *)
	fbAckRTrig						:R_TRIG;			(* Nyugta élképzés *)
	bAckP							:BOOL;				(* Nyugta impulzus *)
	bSafetyError					:BOOL;				(* Safety PLC hiba *)
	fbDoor							:FB_Door;			(* Ajtókör vezérlés *)
	bGlobalEHA						:BOOL;				(* Error-handling active - Hibafigyelés aktív*)
	bError							:BOOL;				(* Globális hiba bit *)
	bDoorOpenReq					:BOOL;				(* Ajtónyitás kérés *)
	sDoorState						:STRING;			(* Ajtó állapot *)
	bUserAdmin						:BOOL;				(* Adminisztrátor bejelentkezve *)
	bUserMaintenance				:BOOL;				(* Karbantartó bejelentkezve *)
	bInitTCPIP						:BOOL := TRUE;
	bFirstCycle						:BOOL := TRUE;
	fbSmartLight					:FB_SmartLight;
	bAirPressError					:BOOL;
	arrEcatSlaveInfo				:ARRAY [0..iSLAVEADDR_ARR_SIZE] OF ST_SlaveStateInfo;
	nSlaveNr						:UINT;
	stSlaveInfo						:ST_SlaveStateInfo;
	fbWorkLight						:FB_WorkLight;
	fbStartAutClient				:NT_StartProcess;
	
(* P1 Camera *)
	fbP1RFID						:Fb_BISM;
	fbP1Lift						:FB_Bistabil;
	fbP1AxisX						:FB_Motor;	
	fbP1AxisY						:FB_Motor;
	fbP1AxisZ						:FB_Motor;
	fbP1PalletDataExchange			:FB_ADSHandler;
	stP1PalletData					:ST_PalletData;
	fbP1FullCycleTime				:FB_FullCycleTime;
	nP1ScrapCounter					:INT;
	bP1ScrapRepeatError				:BOOL;
	stCam1_IN						:ST_Camera_IN;
	stCam1_OUT						:ST_Camera_OUT;	
	fbP1Cam1						:FB_Kamino;

	(* MES *)
	fbP1MesInterface				:FB_MES_INTERFACE_V2;
	bP1MesInitOK					:BOOL := FALSE;
	stP1MesResp						:ST_REQUEST;
	eP1GapFillerCheck_Result		:E_TEST_STATE;
	stP1MesOpState					:ST_GET_OP_STATE;
	stP1MrtMaterial					:ST_MATERIAL;
	stP1NcDat						:ST_MESDAT;
	fbP1ReceipeList					:FB_ReceipeList;


(* P2 Robot *)
	fbP2RFID						:Fb_BISM;
	fbP2Lift						:FB_Bistabil;
	fbP2PalletDataExchange			:FB_ADSHandler;
	stP2PalletData					:ST_PalletData;
	fbP2KRC4						:FB_KRC4;
	fbP2FullCycleTime				:FB_FullCycleTime;
	nP2ScrapCounter					:INT;
	bP2ScrapRepeatError				:BOOL;

	(* MES *)
	fbP2MesInterface				:FB_MES_INTERFACE_V2;
	bP2MesInitOK					:BOOL := FALSE;
	stP2MesResp						:ST_REQUEST;
	eP2Assy_Auto2_Result			:E_TEST_STATE;
	sP2Assy_Auto2_Recipe			:STRING;
	stP2MrtInventoryList			:ST_INVENTORY_LIST;
	stP2Assy_Auto2_OpState			:ST_GET_OP_STATE;
	stP2NcDat						:ST_MESDAT;

(* Stopper *)
	fbP0Stopper						:FB_Stopper;		(* Állomás elötti stopper *)
	fbP1Stopper						:FB_Stopper;		(* P1 kamera pozíció *)
	fbP2Stopper						:FB_Stopper;		(* P2 Robot pozíció *)

(* Conveyor *)
	fbConveyor_1					:FB_Conveyor;		(* Szalag hajtás K41 *)
	fbConveyor_2					:FB_Conveyor;		(* Szalag hajtás K42 *)
	bConveyorsOk					:BOOL;
	bConveyorsErr					:BOOL;

(* Teszt változót *)
	bAdsInfoNextStation				:BOOL;
	fbPalletDataExchange			:FB_ADSHandler;
	stPalletData					:ST_PalletData;

END_VAR

// ---- GVLs/GVL_Persistenet.TcGVL
VAR_GLOBAL PERSISTENT
	sST10_NetId				:STRING;						// Local 192.168.102.101.1.1
	bMesEnable				:BOOL;							// MES rendszer engedélyezése
	bTechEMYStopIgnored		:BOOL;							// Technológiai Vészstop kikapcsolása
	arrCamSeq				:ARRAY [1..64] OF ST_CamSeq;
	rVelocity				:REAL;
	nWorkLightTime			:UINT;
END_VAR

// ---- GVLs/GVL_Recipe.TcGVL
VAR_GLOBAL
	arrP1RecipeNames		:ARRAY[1..200] OF STRING;
	stP1Recipe				:ST_SCR_RECIPE;
	fbP1RecipeManager		:FB_RecipeManager;	

	bP1RecipeLoad			:BOOL;
	bP1RecipeSave			:BOOL;
	bP1RecipeRefresh		:BOOL;
	nP1RecipeIdx			:INT := 1;
	sP1RecipeName			:STRING (1000);
END_VAR

// ---- GVLs/GVL_Safety.TcGVL
VAR_GLOBAL
	i_bKukaEstopBtn		AT %I*		:BOOL;			// Kuka vészgomb státusz
	i_bGreenBtn			AT %I*		:BOOL;			// Master On nyomógomb

	
	(* Digital input AS1*)
	i_bEmyStopBtn1		AT %I*		:BOOL;			// I1.1
	i_bEmyStopBtn2		AT %I*		:BOOL;			// I1.2
	i_bDoor1Open		AT %I*		:BOOL;			// I1.3
	i_bDoor2Open		AT %I*		:BOOL;			// I1.4
	i_bDoor3Open		AT %I*		:BOOL;			// I1.5
	i_bDoor4Open		AT %I*		:BOOL;			// I1.6
	i_bLO1EDM			AT %I*		:BOOL;			// I1.7
	i_bLO2EDM			AT %I*		:BOOL;			// I1.8
													// I1.9
													// I1.10
	i_bRedBtn			AT %I*		:BOOL;			// I1.11
													// I1.12
													// ...
													// I1.16
													
	i_bSafetyFbErr		AT %I*		:BOOL;			// Safety hiba
	i_bSafetyComErr		AT %I*		:BOOL;			// Safety hiba
	i_bSafetyOtherErr	AT %I*		:BOOL;			// Safety hiba
	i_bSafetyLO1EDMErr	AT %I*		:BOOL;			// EDM hiba
	i_bSafetyLO2EDMErr	AT %I*		:BOOL;			// EDM hiba

	i_bAX5805ErrorX		AT %I*		:BOOL;	
	i_bAX5805ErrorY		AT %I*		:BOOL;	
	i_bAX5805ErrorZ		AT %I*		:BOOL;	
	
	i_bEmyOK			AT %I*		:BOOL;
	i_bDoorOK			AT %I*		:BOOL;

	
	q_bSafety_Run		AT %Q*		:BOOL;	
	q_bSafety_Reset		AT %Q*		:BOOL;	
	q_bSafety_Ack		AT %Q*		:BOOL;
	q_bAX5805_Ack		AT %Q*		:BOOL;	
	q_bLO1EDM			AT %Q*		:BOOL;
	q_bLO2EDM			AT %Q*		:BOOL;
END_VAR

// ---- POUs/MAIN.TcPOU
PROGRAM MAIN
VAR
//	fbEventlogger				:FB_TcEventLogger;	// Elvégzi az FB_EVENTHANDLER 
	aErrorActive				:ARRAY[1..nNbrOfAlarms] OF WORD;
	aErrorID1					:ARRAY[1..nNbrOfAlarms] OF STRING(255);
	aErrorID2					:ARRAY[1..nNbrOfAlarms] OF STRING(255);
	afbAlarms					:ARRAY[1..nNbrOfAlarms] OF FB_TcAlarm;
	i							:UINT;
	fbAirTimer					:TON;
	fbUPS						:FB_UpsC69xx;
	bConsolTest					:bool;
END_VAR

IF bFirstCycle THEN Init(); END_IF
IF NOT bP1MesInitOK OR NOT bP2MesInitOK THEN Init_MES(); END_IF
Alarm();
Blink();
Conveyor();
Door();
Light();
Mode();
Safety();

P1_Camera();
P1_Camera.Recipe();
P1_Camera.Camera();
P1_Camera.DataExchange();
P1_Camera.RFID();
P1_Camera.Pneu();
P1_Camera.Servo();
P1_Camera.MES();
P1_Camera.Diag();

P2_Robot();
P2_Robot.KRC4();
P2_Robot.DataExchange();
P2_Robot.RFID();
P2_Robot.Pneu();
P2_Robot.MES();
P2_Robot.Diag();

Diag();
Harman_AutClient();
MesTest();

fbUPS(
	bEnable:= TRUE, 
	tShdnTime:= T#5S, 
	nShdnDelay:= 0, 
	bPowerOK=> , 
	nBatteryLife=> , 
	bError=> , 
	nErrId=> );
	
fbPalletDataExchange(
	stPalletData:= stPalletData, 
	sName:= 'Paletta adatok', 
	bAck:= bAckP, 
	sAMSNetId:= sST10_NetId, 
	stEventEntry:= TC_EVENTS.MyEvent.fbPalletDataExchange);

IF fbPalletDataExchange.bDone AND fbPalletDataExchange.eCommand <> NoCmd THEN
	fbPalletDataExchange.eCommand := NoCmd;
END_IF

ACTION Alarm:
// Hibakezelés
fbAckRTrig(CLK:= bAckHMI OR i_bRedBtn, Q=> bAckP);

IF fbAckRTrig.Q THEN
	bAckHMI := FALSE;
END_IF

(* Collect global error *)
bError :=	bAirPressError OR
			P1_Camera.stPos.bError OR
			P2_Robot.stPos.bError OR
			bConveyorsErr OR
			bSafetyError OR
			bP1ScrapRepeatError OR
			bP2ScrapRepeatError;
			
(* Air pressure error *)
fbAirTimer(IN:= i_bEMYOK AND NOT i_bAirOk, PT:= T#10S, Q=> bAirPressError);

(* Scrap repeat error *)
bP1ScrapRepeatError :=	nP1ScrapCounter > 3;
bP2ScrapRepeatError :=	nP2ScrapCounter > 3;

IF bAckP AND (bP1ScrapRepeatError OR bP2ScrapRepeatError) THEN
	nP1ScrapCounter := 0;
	nP2ScrapCounter := 0;
END_IF

(* General errors *)
aErrorActive[1].0 := bAirPressError;
aErrorActive[2].0 := i_bSafetyComErr;
aErrorActive[3].0 := i_bSafetyFbErr;
aErrorActive[4].0 := i_bSafetyOtherErr;
aErrorActive[5].0 := i_bSafetyLO1EDMErr;
aErrorActive[6].0 := i_bSafetyLO2EDMErr;
aErrorActive[7].0 := i_bAX5805ErrorX;
aErrorActive[8].0 := i_bAX5805ErrorY;
aErrorActive[9].0 := i_bAX5805ErrorZ;
aErrorActive[10].0 := NOT i_bDC1OK;
aErrorActive[11].0 := NOT i_bDC2OK;
aErrorActive[12].0 := bP1ScrapRepeatError;
aErrorActive[13].0 := bP2ScrapRepeatError;



FOR i := 1 TO nNbrOfAlarms DO
	IF aErrorActive[i].0 THEN
		IF (afbAlarms[i].eConfirmationState <> 2 AND afbAlarms[i].nTimeCleared <> 0 AND afbAlarms[i].nTimeConfirmed <> 0) OR //Ha már volt alarm, akkor van bennük érték
			(afbAlarms[i].eConfirmationState = 1 AND afbAlarms[i].nTimeCleared = 0 AND afbAlarms[i].nTimeConfirmed = 0)	//Első futás esetén
		THEN
			IF aErrorActive[i].1 AND aErrorActive[i].2 THEN
				afbAlarms[i].ipArguments.Clear().AddString(aErrorID1[i]).AddString(aErrorID2[i]);
			ELSIF aErrorActive[i].1 THEN
				afbAlarms[i].ipArguments.Clear().AddString(aErrorID1[i]);
			ELSE
				afbAlarms[i].ipArguments.Clear();
			END_IF
			afbAlarms[i].Raise(0);
		END_IF	
	ELSE
		IF (afbAlarms[i].eConfirmationState = 2 OR afbAlarms[i].eConfirmationState = 3) AND afbAlarms[i].nTimeCleared = 0 THEN
			afbAlarms[i].Clear(0, FALSE);
		END_IF		
	END_IF
END_FOR
END_ACTION

ACTION Door:
fbDoor.bDoorsClosed := NOT	(i_bDoor1Open OR
							i_bDoor2Open OR 
							i_bDoor3Open OR 
							i_bDoor4Open); 
							
fbDoor(
	bDoorButton:= i_bDoorOpenBtn, 
	bOpenEnable:= P1_Camera.stPos.bDoorOpenEnable AND P2_Robot.stPos.bDoorOpenEnable, 
	bDoorsClosed:= , 
	bDoorsLocked:= i_bDoorOK, 
	bBlink:= bBL100p100, 
	bCloseOut=> q_bLockDoor, 
	bDoorButtonLED=> q_bWhiteBtnLed, 
	bObenRequestOut=> bDoorOpenReq);
END_ACTION

ACTION Harman_AutClient:
fbStartAutClient(
	NETID:= '192.168.102.141.1.1', 
	PATHSTR:= 'C:\tozsolti\ConsoleApp1.exe', 
	DIRNAME:= 'C:\tozsolti', 
	COMNDLINE:= 'ConsoleApp1.exe', 
	START:= bConsolTest, 
	TMOUT:= T#1S, 
	BUSY=> , 
	ERR=> , 
	ERRID=> );
END_ACTION

ACTION Init:
	(* Bind errors *)
afbAlarms[1].CreateEx(TC_Events.MyEvent.Gen_1, TRUE, 0);
afbAlarms[2].CreateEx(TC_Events.MyEvent.Gen_2, TRUE, 0);
afbAlarms[3].CreateEx(TC_Events.MyEvent.Gen_3, TRUE, 0);
afbAlarms[4].CreateEx(TC_Events.MyEvent.Gen_4, TRUE, 0);
afbAlarms[5].CreateEx(TC_Events.MyEvent.Gen_5, TRUE, 0);
afbAlarms[6].CreateEx(TC_Events.MyEvent.Gen_6, TRUE, 0);
afbAlarms[7].CreateEx(TC_Events.MyEvent.Gen_7, TRUE, 0);
afbAlarms[8].CreateEx(TC_Events.MyEvent.Gen_8, TRUE, 0);
afbAlarms[9].CreateEx(TC_Events.MyEvent.Gen_9, TRUE, 0);
afbAlarms[10].CreateEx(TC_Events.MyEvent.Gen_10, TRUE, 0);
afbAlarms[11].CreateEx(TC_Events.MyEvent.Gen_11, TRUE, 0);
afbAlarms[12].CreateEx(TC_Events.MyEvent.Gen_12, TRUE, 0);

fbP2KRC4.stEventArray[0] := TC_EVENTS.MyEvent.fbP2KRC4_Alarm0;
fbP2KRC4.stEventArray[1] := TC_EVENTS.MyEvent.fbP2KRC4_Alarm1;
fbP2KRC4.stEventArray[2] := TC_EVENTS.MyEvent.fbP2KRC4_Alarm2;
fbP2KRC4.stEventArray[3] := TC_EVENTS.MyEvent.fbP2KRC4_Alarm3;
fbP2KRC4.stEventArray[4] := TC_EVENTS.MyEvent.fbP2KRC4_Alarm4;
fbP2KRC4.stEventArray[5] := TC_EVENTS.MyEvent.fbP2KRC4_Alarm5;
fbP2KRC4.stEventArray[6] := TC_EVENTS.MyEvent.fbP2KRC4_Alarm6;
fbP2KRC4.stEventArray[7] := TC_EVENTS.MyEvent.fbP2KRC4_Alarm7;

bFirstCycle := False;
END_ACTION

ACTION Init_MES:
IF NOT bP1MesInitOK THEN
	IF fbP1MesInterface.LOCAL_INIT_SERVICE() THEN
		bP1MesInitOK := TRUE;
	END_IF
END_IF

IF bP1MesInitOK AND NOT bP2MesInitOK THEN
	IF fbP2MesInterface.REMOTE_INIT_SERVICE() THEN
		bP2MesInitOK := TRUE;
	END_IF
END_IF
END_ACTION

ACTION Light:
fbSmartLight(
	bEmyStop:= i_bEmyStopBtn1 OR i_bEmyStopBtn2, 
	bEmyOK:= i_bEmyOK, 
	bError:= bError, 
	bOutOfStock:= FALSE);
	
// Piros jelzés
IF i_bEmyStopBtn1 OR i_bEmyStopBtn2 THEN
	q_bRedBtnLed := TRUE;
ELSE
	IF bError THEN
		q_bRedBtnLed := bBL500p500;
	ELSIF P1_Camera.stPos.nState = 100100 THEN
		q_bRedBtnLed := FALSE;
	ELSE
		q_bRedBtnLed := FALSE;
	END_IF
END_IF

// Zöld jelzés
IF i_bEmyStopBtn1 OR i_bEmyStopBtn2 THEN
	q_bGreenBtnLed := FALSE;
ELSE
	IF i_bEmyOK THEN
		q_bGreenBtnLed := TRUE;
	ELSE
		q_bGreenBtnLed := bBL500p500;
	END_IF
END_IF

// Munkatér világítás
IF nWorkLightTime > 120 THEN nWorkLightTime := 120; END_IF
IF nWorkLightTime < 1 THEN nWorkLightTime := 1; END_IF

fbWorkLight(
		bDoorClose:= fbDoor.bDoorsClosed,
		bManualCtrl:= ,
		nEcoTime:= nWorkLightTime,
		bLightCtrl=> q_bAreaLighting);	
		

															// A cella gyártóképes ha:
q_bST40_Status.0		 :=	i_bEmyOK AND					// vészkör endben
							i_bAirOK AND					// levegő rendben
							i_bDoorOK AND					// ajtók reteszelve
							NOT bManualMode AND				// nincs szervíz üzem
							NOT bStepMode AND				// nincs léptető mód
							fbP2KRC4.RobotIn.Status.bExt;	// a robot ext-be van kapcsolva

q_bST40_Status.8 := bError;									// hiba bit küldése
q_bST40_Status.9 := FALSE;									// anyag kifogyás küldése
END_ACTION

ACTION Mode:
// Üzemmód állítás
IF bManualModeRequest THEN
	IF (P1_Camera.stPos.nState = 0 OR P1_Camera.stPos.nState = 10000 OR P1_Camera.stPos.nState = 150000 OR P1_Camera.stPos.nState >= 200000) AND
		(P2_Robot.stPos.nState = 0 OR P2_Robot.stPos.nState = 10000 OR P2_Robot.stPos.nState = 150000 OR P2_Robot.stPos.nState >= 200000)
	THEN
		sMode := 'Kézi mód';
		nMode := 2;
		bManualMode := TRUE;
		bGlobalEHA := FALSE;
	ELSE
		sMode := 'Kézi mód kérés';
		nMode := 1;
	END_IF
ELSE
	sMode := 'Automata mód';
	nMode := 0;
	bManualMode := FALSE;
	bGlobalEHA := TRUE;
END_IF

// Léptetés üzem teszteléshez
rtStep(CLK:= bStepHMI or i_bGreenBtn, Q=> bStepP);
IF bStepMode AND bStepP OR NOT bStepMode THEN
	bStepEnable := TRUE;
ELSE
	bStepEnable := FALSE;
END_IF
END_ACTION

ACTION Safety:
(*-----=== Safety GroupPort Run ===-----*)
IF bTechEMYStopIgnored THEN
	q_bSafety_Run := TRUE;
ELSE
	q_bSafety_Run := i_bST10_TechEMYStopOn AND i_bST10_TechEMYStopOn_Quality <= 2000;		// 200ms adatkimaradás is technológiai stop! 	
END_IF

(*-----=== Technológiai vészstop figyelembevételének állapota ===-----*)
q_bST40_TechEMYStopIgnored := bTechEMYStopIgnored;

(*-----=== EDM jelek másolása ===-----*)
q_bLO1EDM := i_bLO1EDM;
q_bLO2EDM := i_bLO2EDM;

(*-----=== Hibakezelés ===-----*)
q_bSafety_Reset := bAckP;
q_bSafety_Ack := bAckP;
q_bAX5805_Ack := bAckP;

bSafetyError :=		i_bSafetyFbErr OR
					i_bSafetyComErr OR
					i_bSafetyOtherErr OR
					i_bSafetyLO1EDMErr OR
					i_bSafetyLO2EDMErr OR
					i_bAX5805ErrorX OR	
					i_bAX5805ErrorY OR	
					i_bAX5805ErrorZ;
END_ACTION

END_PROGRAM

// ---- POUs/FBs/FB_UpsC69xx.TcPOU
FUNCTION_BLOCK FB_UpsC69xx
VAR_INPUT
	bEnable					:BOOL;					// FB Engedély.
	tShdnTime				:TIME := T#10S;			// Tápkimaradási időkorlát
	nShdnDelay				:DWORD := 0;			// Leállítási késleltetés
END_VAR
VAR_OUTPUT
	bPowerOK				:BOOL;					// Tápellátás rendben
	nBatteryLife			:DWORD;					// Akkumulátor állapot (százalékba)
	bError					:BOOL;					// Hiba bit
	nErrId					:UDINT;					// Hiba kód
END_VAR
VAR
	fbGetUpsStatus			:FB_GetUPSStatus;
	ntShutdown				:NT_Shutdown;
	tShutdown				:TON;
END_VAR

(*-----=== UPS ===-----*)
(*	--------------------------------------------------------------------------------
	Leírás		:	C69XX CPU Szünetmentes táp kezelés
	Név			:	FB_UpsC69xx
	Módosító	:	Závori Zsolt
	Dátum		:	2019.07.05
	Revízió		:	1.0
	--------------------------------------------------------------------------------
	Feltételek	:	Tc2_Utilities-(REF), Tc2_IoFunctions
	Változók	:	-
	Visu		:	-
	UserControl	:	-
	--------------------------------------------------------------------------------
	Részletek	:	-					
*)
fbGetUpsStatus(bEnable:= bEnable );
fbGetUpsStatus( 
	bEnable:= bEnable, 
	bError=> bError, 
	nErrId=> nErrId);

nBatteryLife := fbGetUpsStatus.stStatus.BatteryLifePercent;

tShutdown(
		IN:= fbGetUpsStatus.stStatus.ePowerStatus = PowerOnBattery AND
			 fbGetUpsStatus.bValid AND NOT fbGetUpsStatus.bError AND bEnable,
		PT:= tShdnTime);

bPowerOK := (fbGetUpsStatus.stStatus.ePowerStatus = PowerOnLine);		
IF tShutdown.Q THEN
	ntShutdown(
			DELAY:= nShdnDelay, 
			START:= TRUE);
END_IF

END_FUNCTION_BLOCK

// ---- POUs/Blink.TcPOU
PROGRAM Blink
VAR
	tBL1					:FB_GenPulse; (*50ms/50ms*)
	tBL2					:FB_GenPulse; (*100ms/100ms*)
	tBL3					:FB_GenPulse; (*250ms/250ms*)
	tBL4					:FB_GenPulse; (*500ms/500ms*)
	tBL5					:FB_GenPulse; (*1000ms/1000ms*)
	tBL6					:FB_GenPulse; (*750ms/250ms*)
	rtBL1,rtBL2,rtBL3,rtBL4	:R_TRIG;
END_VAR

tBl1(ENQ:= TRUE, PTH:=  T#50MS, PTL:= T#50MS, Q=>GVL_Main.bBL50p50 );
tBl2(ENQ:= TRUE, PTH:=  T#100MS, PTL:= T#100MS, Q=>GVL_Main.bBL100p100 );
tBl3(ENQ:= TRUE, PTH:=  T#250MS, PTL:= T#250MS, Q=>GVL_Main.bBL250p250 );
tBl4(ENQ:= TRUE, PTH:=  T#500MS, PTL:= T#500MS, Q=>GVL_Main.bBL500p500 );
tBl5(ENQ:= TRUE, PTH:=  T#1000MS, PTL:= T#1000MS, Q=>GVL_Main.bBL1000p1000 );
tBl6(ENQ:= TRUE, PTH:=  T#250MS, PTL:= T#750MS, Q=>GVL_Main.bBL250p750 );
rtBL1(CLK:=GVL_Main.bBL50p50, Q=> GVL_Main.bTakt100ms);
rtBL2(CLK:=GVL_Main.bBL100p100, Q=> GVL_Main.bTakt200ms);
rtBL3(CLK:=GVL_Main.bBL250p250, Q=> GVL_Main.bTakt500ms);
rtBL4(CLK:=GVL_Main.bBL500p500, Q=> GVL_Main.bTakt1s);

IF GVL_Main.bTakt100ms THEN
	GVL_Main.nLifeSignal := GVL_Main.nLifeSignal + 1;	
END_IF

IF GVL_Main.nLifeSignal>100 THEN
	GVL_Main.nLifeSignal:=0;
END_IF

END_PROGRAM

// ---- POUs/Conveyor.TcPOU
PROGRAM Conveyor
VAR

END_VAR

(* Szalaghajtások automatikus indítása *)
IF i_bEmyOK AND NOT bManualMode THEN
	fbConveyor_1.bConveyorOnL := TRUE;	
	fbConveyor_1.bConveyorOnR := FALSE;	
	fbConveyor_2.bConveyorOnL := TRUE;	
	fbConveyor_2.bConveyorOnR := FALSE;	

END_IF

(* Szalaghajtások vezérlése *)
fbConveyor_1(
	sName:= 'K41', 
	bEn:= i_bEmyOK, 
	bEHA:= TRUE, 
	bDisableManualCmd:= NOT bManualMode, 
	bAck:= bAckP, 
	stStartEvent:= TC_EVENTS.MyEvent.fbConv1_Start,
	stRunEvent:= TC_EVENTS.MyEvent.fbConv1_Run);

fbConveyor_2(
	sName:= 'K42', 
	bEn:= i_bEmyOK, 
	bEHA:= TRUE, 
	bDisableManualCmd:= NOT bManualMode, 
	bAck:= bAckP, 
	stStartEvent:= TC_EVENTS.MyEvent.fbConv2_Start,
	stRunEvent:= TC_EVENTS.MyEvent.fbConv2_Run);

(* Hibaállapot gyűjtése *)	
bConveyorsErr:=	fbConveyor_1.bError OR
				fbConveyor_2.bError;	
	
(* Üzemkész állapot gyűjtése *)
bConveyorsOk :=	(fbConveyor_1.bMotorOn AND NOT fbConveyor_1.bError) AND
				(fbConveyor_2.bMotorOn AND NOT fbConveyor_2.bError);

(* Megakasztók vezérlése *)
fbP0Stopper(
	bNextReady:= fbP1Stopper.bReady, 
	bMotorRun:= bConveyorsOk, 
	tToNextStopper:= T#3S, 
	bStationReady:= TRUE, 
	bStationFinished:= TRUE,
	bReady=> q_bST40_ConveyorReady);
	
fbP1Stopper(
	bNextReady:= fbP2Stopper.bReady, 
	bMotorRun:= bConveyorsOk, 
	tToNextStopper:= T#4.5S, 
	bStationReady:= P1_Camera.stPos.nState = 10000, 
	bStationFinished:= P1_Camera.stPos.nState = 100000);

fbP2Stopper(
	bNextReady:= i_bST51_ConveyorReady, 
	bMotorRun:= bConveyorsOk, 
	tToNextStopper:= T#4.5S, 
	bStationReady:= P2_Robot.stPos.nState = 10000, 
	bStationFinished:= P2_Robot.stPos.nState = 100000);

END_PROGRAM

// ---- POUs/P1_Camera.TcPOU
PROGRAM P1_Camera
VAR
		stPos					:ST_PosData;
		tCycleTime				:TON;
		i						:INT;
		tPalletStartTime		:TON;
		nCycle_Idx				:BYTE;
		arrMES_Temp				:ARRAY [0..2] OF ST_P1MesData;
END_VAR

(*Időzítők***************************************************)
IF (stPos.nState>10000) AND (stPos.nState<100000) AND NOT tCycleTime.Q THEN
	stPos.nCycleTime := TIME_TO_REAL(tCycleTime.ET)/1000;
END_IF
tCycleTime(IN:= (stPos.nState>10000) AND (stPos.nState<150000), PT:= T#200S);							// A palettára várakozás nincs beszámolva
tPalletStartTime(IN:= NOT i_bP2PalletSensor AND fbConveyor_1.bMotorOn, PT:= T#4S);					// Alaphelyzet felvétel késleltetése!

(*Triggerek**************************************************)

(*Vész rendszer**********************************************)
IF	(NOT (i_bEmyOK AND fbDoor.bDoorsLocked) AND stPos.nState > 0) OR									// Nincs vészkör, vagy
	(NOT i_bDoorOK AND (stPos.nState>=60 AND stPos.nState<=1000)) OR									// alaphelyzetfelvétel közbe megszűnik az ajtókör vagy
	(NOT i_bDoorOK AND (stPos.nState>=10060 AND stPos.nState<=100060)) THEN							// folyamat közbe megszűnik az ajtókör 
		stPos.nState := 0;
END_IF;

(*Hibakezelés************************************************)
IF stPos.nState > 0 AND stPos.nState < 150000 THEN
	stPos.nStateLast := stPos.nState;
	IF	fbP1Lift.bError OR
		fbP1PalletDataExchange.bError OR
		(fbP1AxisX.bError AND i_bDoorOK (*AND stP1.nState >= 500*)) OR
		(fbP1AxisY.bError AND i_bDoorOK (*AND stP1.nState >= 500*)) OR
		(fbP1AxisZ.bError AND i_bDoorOK (*AND stP1.nState >= 500*)) OR
		stPos.bError THEN
			stPos.nState := 200000;
	END_IF
END_IF

(*Engedélyek *************************************************)
IF stPos.nState <= 10000
	OR stPos.nState = 100000
	OR stPos.nState = 150000
	OR stPos.nState >= 200000
THEN
	stPos.bManualModeEnable := TRUE;
ELSE
	stPos.bManualModeEnable := FALSE;
END_IF

IF stPos.nState = 0
	OR stPos.nState = 10000
	OR stPos.nState = 100000
	OR stPos.nState = 150000
	OR stPos.nState >= 200000
THEN
	stPos.bDoorOpenEnable := TRUE;
ELSE
	stPos.bDoorOpenEnable := FALSE;
END_IF

(*Kézi üzem *************************************************)
IF bManualMode THEN
	stPos.nState := 150000;
END_IF

(*Automata üzem *********************************************)
CASE stPos.nState OF
{region "Init process"}
	0:		stPos.sState := CONCAT(UDINT_TO_STRING(stPos.nState) ,' - Vészkör vagy ajtókör bontva - Működtetések törlése');
			fbP1AxisX.bGoPosition := FALSE;
			fbP1AxisY.bGoPosition := FALSE;
			fbP1AxisZ.bGoPosition := FALSE;
			fbP1Lift.bBasePosCmd := TRUE;
			fbP1Lift.bWorkPosCmd := FALSE;
			fbP1PalletDataExchange.eCommand := NoCmd;
			stPos.bError := FALSE;
			stPos.nErrorCode := 0;
			IF i_bDoorOK THEN
				IF bStepEnable THEN
					stPos.nState := stPos.nState + 20;
				END_IF
			END_IF
			
	20:		stPos.sState := CONCAT(UDINT_TO_STRING(stPos.nState) ,' - Alaphelyzetfelvétel - Kiemelő alaphelyzetbe');
			fbP1Lift.bBasePosCmd := TRUE;
			fbP1Lift.bWorkPosCmd := FALSE;
			IF fbP1Lift.bBasePosStab THEN
				IF bStepEnable THEN
					stPos.nState := stPos.nState + 20;
				END_IF
			END_IF
			
	40:		stPos.sState := CONCAT(UDINT_TO_STRING(stPos.nState) ,' - AX5805 safety ellenőrzés');	
			IF (i_bAX5805ErrorX OR i_bAX5805ErrorX) AND NOT q_bAX5805_Ack THEN
				q_bAX5805_Ack := TRUE;
			ELSIF NOT (i_bAX5805ErrorX OR i_bAX5805ErrorY OR i_bAX5805ErrorZ) THEN
				q_bAX5805_Ack := FALSE;
				IF bStepEnable THEN
					stPos.nState := stPos.nState + 20;
				END_IF
			END_IF

	60:		stPos.sState := CONCAT(UDINT_TO_STRING(stPos.nState) ,' - Szervo X tengely drive ellenőrzés');	
			IF NOT fbP1AxisX.Axis.Status.DriveDeviceError THEN
				IF bStepEnable THEN
					stPos.nState := stPos.nState + 20;
				END_IF
			END_IF

	80:		stPos.sState := CONCAT(UDINT_TO_STRING(stPos.nState) ,' - Szervo X tengely NC ellenőrzés');	
			IF NOT fbP1AxisX.Axis.Status.Error THEN
				IF bStepEnable THEN
					stPos.nState := stPos.nState + 20;
				END_IF
			END_IF

	100:	stPos.sState := CONCAT(UDINT_TO_STRING(stPos.nState) ,' - Szervo X tengely ellenőrzés');	
			IF fbP1AxisX.nState = 1000 THEN
				IF bStepEnable THEN
					stPos.nState := stPos.nState + 20;
				END_IF
			END_IF
			
	120:	stPos.sState := CONCAT(UDINT_TO_STRING(stPos.nState) ,' - Szervo Y tengely drive ellenőrzés');	
			IF NOT fbP1AxisY.Axis.Status.DriveDeviceError THEN
				IF bStepEnable THEN
					stPos.nState := stPos.nState + 20;
				END_IF
			END_IF

	140:	stPos.sState := CONCAT(UDINT_TO_STRING(stPos.nState) ,' - Szervo Y tengely NC ellenőrzés');	
			IF NOT fbP1AxisY.Axis.Status.Error THEN
				IF bStepEnable THEN
					stPos.nState := stPos.nState + 20;
				END_IF
			END_IF

	160:	stPos.sState := CONCAT(UDINT_TO_STRING(stPos.nState) ,' - Szervo Y tengely ellenőrzés');	
			IF fbP1AxisY.nState = 1000 THEN
				IF bStepEnable THEN
					stPos.nState := stPos.nState + 20;
				END_IF
			END_IF

	180:	stPos.sState := CONCAT(UDINT_TO_STRING(stPos.nState) ,' - Szervo Z tengely drive ellenőrzés');	
			IF NOT fbP1AxisZ.Axis.Status.DriveDeviceError THEN
				IF bStepEnable THEN
					stPos.nState := stPos.nState + 20;
				END_IF
			END_IF

	200:	stPos.sState := CONCAT(UDINT_TO_STRING(stPos.nState) ,' - Szervo Z tengely NC ellenőrzés');	
			IF NOT fbP1AxisZ.Axis.Status.Error THEN
				IF bStepEnable THEN
					stPos.nState := stPos.nState + 20;
				END_IF
			END_IF

	220:	stPos.sState := CONCAT(UDINT_TO_STRING(stPos.nState) ,' - Szervo Z tengely ellenőrzés');	
			IF fbP1AxisZ.nState = 1000 THEN
				IF bStepEnable THEN
					stPos.nState := 500;
				END_IF
			END_IF
	 
			
	500:	stPos.sState := CONCAT(UDINT_TO_STRING(stPos.nState) ,' - Z tengely alaphelyzetbe mozgatása');			
			fbP1AxisZ.rPosition1 := 0;
			fbP1AxisZ.rVelocity1 := 100;
			fbP1AxisZ.bGoPosition := TRUE;
			IF fbP1AxisZ.bDone THEN
				IF bStepEnable THEN
					fbP1AxisZ.bGoPosition := FALSE;
					stPos.nState := stPos.nState + 20;
				END_IF
			END_IF
			
	520:	stPos.sState := CONCAT(UDINT_TO_STRING(stPos.nState) ,' - X tengely alaphelyzetbe mozgatása');			
			fbP1AxisX.rPosition1 := 0;
			fbP1AxisX.rVelocity1 := 100;
			fbP1AxisX.bGoPosition := TRUE;
			IF fbP1AxisX.bDone THEN
				IF bStepEnable THEN
					fbP1AxisX.bGoPosition := FALSE;
					stPos.nState := stPos.nState + 20;
				END_IF
			END_IF
			
	540:	stPos.sState := CONCAT(UDINT_TO_STRING(stPos.nState) ,' - Y tengely alaphelyzetbe mozgatása');			
			fbP1AxisY.rPosition1 := 0;
			fbP1AxisY.rVelocity1 := 100;
			fbP1AxisY.bGoPosition := TRUE;
			IF fbP1AxisY.bDone THEN
				IF bStepEnable THEN
					fbP1AxisY.bGoPosition := FALSE;
					stPos.nState := stPos.nState + 20;
				END_IF
			END_IF
					 
	560:	stPos.sState := CONCAT(UDINT_TO_STRING(stPos.nState) ,' - Várakozás paletta mozgásra a pzíciók között');
			IF tPalletStartTime.Q THEN									// Normál esetben nem kerülhet ebbe az állapotba a berendezés!
				IF bStepEnable THEN										// Ha viszont P1 elengedi a palettát, amin jó termék van, és az még nem érkezik meg P2-be
					stPos.nState := 10000;								// a következő paletta ami üres megérkezik P1-be, ekkor nyomnak egy vészstopot, kinyitják az ajtót és visszahúzzák
				END_IF													// a palettát P2 elől, akkor induláskor P1 rögtön elengedné az üres palettát igy P2-be 2 paletta érkezne!!!!
			END_IF														// Ebből a hibából automatikusan csak selejtezéssel lehetne kiszedni az állomást!!! Ez nem lenne túl szerencsés!!

{endregion}
			
(* Alaphelyzet *********************************************************************)
	10000:	stPos.sState := CONCAT(UDINT_TO_STRING(stPos.nState) ,' - Alaphelyzet, termékre vár');
			IF fbP1RFID.bTagPresent AND fbP1Stopper.bPalletAtStopper AND NOT bP1ScrapRepeatError THEN
				IF bStepEnable THEN
					stPos.nState := stPos.nState + 20;
				END_IF
			END_IF	

{region "Pallet receive"}
	(*-----=== Hordozólap adatok lekérdezése ST10-től ===-----*)
	10020:	stPos.sState := CONCAT(UDINT_TO_STRING(stPos.nState) ,' - Paletta adatok lekérdezése');
			fbP1PalletDataExchange.nIndex := fbP1RFID.nTAGData;
			IF bStepEnable THEN
				fbP1PalletDataExchange.eCommand := Read;
				stPos.nState := stPos.nState + 20;
			END_IF
			
	(*-----=== Hordozólap adatok lekérdezése ST10-től ===-----*)
	10040:	stPos.sState := CONCAT(UDINT_TO_STRING(stPos.nState) ,' - Paletta adatok lekérdezése');
			IF fbP1PalletDataExchange.bDone AND NOT fbP1PalletDataExchange.bError THEN
				IF bStepEnable THEN
					fbP1PalletDataExchange.eCommand := NoCmd;
					stPos.nState := stPos.nState + 20;
				END_IF
			END_IF

	(*-----=== Hordozólap adatok kiértékelése ===-----*)
	10060:	stPos.sState := CONCAT(UDINT_TO_STRING(stPos.nState) ,' - Paletta adatok lekérdezése');
			IF		stP1PalletData.nPalletState = 2 AND			// OK termék a palettán
					stP1PalletData.nDone.3 AND					// Diszpenzálás kész
					NOT stP1PalletData.nDone.4 THEN				// Kamerás ell. még nincs kész
						IF bStepEnable THEN						// Mehet a kiemelés -> Normál folyamat
							nCycle_Idx := 0;

							arrMES_Temp[0].nOP_Index := nP1GapFillerCheckCover_Index;
							arrMES_Temp[0].sDMC_Code := stP1PalletData.sCoverCode;
							arrMES_Temp[0].sOP_Name := 'OP_GAP_FILLER_CHK_COVER';
							
							arrMES_Temp[1].nOP_Index := nP1CheckSim_Index;
							arrMES_Temp[1].sDMC_Code := stP1PalletData.sMRTCode;
							arrMES_Temp[1].sOP_Name := 'OP_CHECK_SIM';
	
							arrMES_Temp[2].nOP_Index := nP1CheckComponent_Index;
							arrMES_Temp[2].sDMC_Code := stP1PalletData.sMRTCode;
							arrMES_Temp[2].sOP_Name := 'OP_CHECK_COMPONENT';
	
							stPos.nState := stPos.nState + 20;
						END_IF
			ELSIF	stP1PalletData.nPalletState = 41 THEN		// Teszt hordozólap a kamerához
						IF bStepEnable THEN						// Még nincs funkció -> Tovább engedés
							stPos.nState := 96060; //????
						END_IF
			ELSIF	stP1PalletData.nPalletState = 2 AND			// OK termék a palettán
					NOT stP1PalletData.nDone.3 THEN				// Diszpenzálás nincs kész !
						IF bStepEnable THEN						// Átemelt hordozólap!?!? -> Selejtezés
							stP1PalletData.nPalletState := 1;
							stP1PalletData.nDone.4	:= TRUE;
							stP1PalletData.nErrorCode := 4100;
							stPos.nState := 96000;
						END_IF
			ELSIF	stP1PalletData.nPalletState = 1 THEN		// Selejt termék a palettán
						IF bStepEnable THEN						// Nincs kiemelés -> Tovább engedés
							stPos.nState := 96060;
						END_IF
			ELSIF	stP1PalletData.nPalletState = 0 THEN		// Üres paletta
						IF bStepEnable THEN						// Nincs kiemelés -> Tovább engedés
							stPos.nState := 96060;
						END_IF
			ELSE												// Nincs teendő, más állomásnak szánt hordozólap
						IF bStepEnable THEN						// Nincs kiemelés -> Tovább engedés
							stPos.nState := 96060;
						END_IF			
			END_IF

	(*-----=== MES engedély ellenőrzése ===-----*)
	10080:	stPos.sState := CONCAT(UDINT_TO_STRING(stPos.nState) ,' - MES engedély ellenőrzése');
			IF bMesEnable THEN
				IF bStepEnable THEN
					stPos.nState := 14000;
				END_IF
			ELSE
				IF bStepEnable THEN
					stPos.nState := 16000;
				END_IF				
			END_IF
{endregion}

{region "Normal process"} 
(*-----=== Recept lista kezelés ===-----*)
(* Get MRT OP state *)
14000:		stPos.sState := CONCAT(UDINT_TO_STRING(stPos.nState) ,' - Get OP state MRT (1026)');
			IF fbP1MesInterface.GET_CURRENT_OPERATION_STATE(stP1PalletData.sMRTCode, 0,stP1MesOpState) THEN
				IF stP1MesResp.RESP_CODE = '0' or stP1MesResp.RESP_CODE = '377'	THEN									// MRT OP state OK
					IF bStepEnable THEN
						stP1MrtMaterial.MATERIAL := stP1MesOpState.MAT_NO;
						stP1MrtMaterial.REVISION := stP1MesOpState.REVISION;
						nCycle_Idx := 0;
						stPos.nState := 14100;
					END_IF		
				ELSE
					IF bStepEnable THEN													// Get OP state hiba
						stP1PalletData.nPalletState := 1;
						stP1PalletData.nDone.4	:= TRUE;
							stP1PalletData.nErrorCode := 4101;
						stPos.nState := 96000;
					END_IF
				END_IF
			END_IF

	 
14100:		stPos.sState := CONCAT(UDINT_TO_STRING(stPos.nState) ,' - Get Material Custom Data (1037)');
			IF fbP1MesInterface.GET_MAT_CUSTOM_DATA(stP1MrtMaterial, 0) THEN
				IF stP1MesResp.RESP_CODE = '0'	THEN									// Get Custom Data OK
					IF bStepEnable THEN
						stPos.nState := stPos.nState + 20;
					END_IF		
				ELSE
					IF bStepEnable THEN													// Get Custom Data hiba
						stP1PalletData.nPalletState := 1;
						stP1PalletData.nDone.4	:= TRUE;
							stP1PalletData.nErrorCode := (4102 + nCycle_Idx);
						stPos.nState := 96000;
					END_IF
				END_IF
			END_IF		  

14120:		stPos.sState := CONCAT(UDINT_TO_STRING(stPos.nState) ,' - Get Custom Data By Key');
			IF fbP1MesInterface.GET_CUSTOM_DATA_BY_KEY(CONCAT(arrMES_Temp[nCycle_Idx].sOP_Name, '_R'), arrMES_Temp[nCycle_Idx].sOP_CustomData) THEN
				IF arrMES_Temp[nCycle_Idx].sOP_CustomData <> ''	THEN					// Get Custom Data by key OK
					IF bStepEnable THEN
						arrMES_Temp[nCycle_Idx].sOP_ReceipeList := arrMES_Temp[nCycle_Idx].sOP_CustomData;
						stPos.nState := stPos.nState + 20;
					END_IF		
				ELSE
					IF bStepEnable THEN													// Get Custom Data by key hiba
						stP1PalletData.nPalletState := 1;
						stP1PalletData.nDone.4	:= TRUE;
							stP1PalletData.nErrorCode := (4103 + nCycle_Idx);
						stPos.nState := 96000;
					END_IF
				END_IF
			END_IF		  

14140:		stPos.sState := CONCAT(UDINT_TO_STRING(stPos.nState) ,' - Recept lista ellenőrzése');   
			IF nCycle_Idx >= 2 THEN
				IF bStepEnable THEN						// Custom fied-ek átemelve -> Gyí, gyí gyí !!!
					nCycle_Idx := 0;
					stPos.nState := 14200;
				END_IF
			ELSE
				IF bStepEnable THEN
					nCycle_Idx := nCycle_Idx + 1;		// Van még háta Custom fiel -> Mehet a köv. lekérdezés
					stPos.nState := 14100;
				END_IF
			END_IF		

14200:
			stPos.nState := 15000;		

				 
(*-----=== MES 3010 (Start SFC) ===-----*)
	15000:	stPos.sState := CONCAT(UDINT_TO_STRING(stPos.nState) ,' - Start SFC (3010)');
			eP1GapFillerCheck_Result := E_TEST_STATE.PASSED;	
			IF fbP1MesInterface.START_SFC(arrMES_Temp[nCycle_Idx].sDMC_Code, arrMES_Temp[nCycle_Idx].nOP_Index) THEN
				IF stP1MesResp.RESP_CODE = '0'	THEN									// Jó termék
					IF bStepEnable THEN
						stPos.nState := stPos.nState + 20;
					END_IF		
				ELSE
					IF bStepEnable THEN													// Selejt
						stP1PalletData.nPalletState := 1;
						stP1PalletData.nDone.4	:= TRUE;
							stP1PalletData.nErrorCode := 4111 + nCycle_Idx;
						stPos.nState := 96000;
					END_IF
				END_IF
			END_IF

(*			// Custom field olvasása miatt kiesik! A receptlistát előre le kell tölteni! 2021.02.15
	15020:	stP1.sState := CONCAT(UDINT_TO_STRING(stP1.nState) ,' - Get recipe name');	
			IF fbP1MesInterface.GET_RECIPE_NAME_BY_OPERATION_JSON(arrMES_Temp[nCycle_Idx].sOP_Name, sP1RecipeName) THEN
			IF sP1RecipeName <>'' THEN
				stP1.nState := 16000;
			ELSE
				stP1PalletData.nPalletState := 1;							// Nincs recept név, viszont az SFC startolva -> le kell zárni hibával.
				stP1PalletData.nDone.4	:= TRUE;
				stP1PalletData.nErrorCode := 4103;
				eP1GapFillerCheck_Result := E_TEST_STATE.FAILED;
				stP1NcDat.MESDAT[stP1NcDat.N].RESPONSE_CODE := '4103';
				stP1NcDat.MESDAT[stP1NcDat.N].RESPONSE_DESCRIPTION := CONCAT(CONCAT('The ',arrMES_Temp[nCycle_Idx].sOP_Name),' recipe missing');
				stP1NcDat.MESDAT[stP1NcDat.N].CLIENT_DATE := fbP1MesInterface.GET_LOCAL_TIME();
				stP1NcDat.MESDAT[stP1NcDat.N].TEST_STATE := INT_TO_STRING(E_TEST_STATE.FAILED);
				stP1NcDat.MESDAT[stP1NcDat.N].TEST_STEP := INT_TO_STRING(stP1NcDat.N);
				stP1NcDat.MESDAT[stP1NcDat.N].VALUE := '0';
				stP1.nState := 95000;
			END_IF
		END_IF
*)

	15020:	stPos.sState := CONCAT(UDINT_TO_STRING(stPos.nState) ,' - Receptnév átadása');	
			fbP1ReceipeList(
				sReceipeListIn:= arrMES_Temp[nCycle_Idx].sOP_ReceipeList,
				sReceipeListOut=> arrMES_Temp[nCycle_Idx].sOP_ReceipeList,
				sReceipe=> sP1RecipeName,
				bEmpty=> );
			stPos.nState := 16000;

(*-----=== Recept kezelés ===-----*)
	16000:	stPos.sState := CONCAT(UDINT_TO_STRING(stPos.nState) ,' - Recept lista frissítése');
			bP1RecipeRefresh := TRUE;
			IF fbP1RecipeManager.DONE AND fbP1RecipeManager.RECIPE_CNT > 0 THEN
				IF bStepEnable THEN
						bP1RecipeRefresh := FALSE;
						stPos.nState := stPos.nState + 20;
				END_IF
			END_IF

	16020:	stPos.sState := CONCAT(UDINT_TO_STRING(stPos.nState) ,' - Várakozás recept lista frissítés befejezésére');
			IF NOT fbP1RecipeManager.DONE AND NOT fbP1RecipeManager.RESET THEN
				IF bMesEnable THEN
					IF bStepEnable THEN
							stPos.nState := stPos.nState + 20;
					END_IF
				ELSE
					IF bStepEnable THEN
							sP1RecipeName := arrP1RecipeNames[nCycle_Idx + 1];			// Kikapcsolt MES esetén is legyen ellenőrzés 
							stPos.nState := stPos.nState + 20;
					END_IF
				END_IF
			END_IF

	16040:	stPos.sState := CONCAT(UDINT_TO_STRING(stPos.nState) ,' - Recept betöltése');
			bP1RecipeLoad := TRUE;
			IF fbP1RecipeManager.DONE THEN
				IF bStepEnable THEN
						bP1RecipeLoad := FALSE;
						i := 0;
						stP1NcDat.N := 1;
						stPos.nState := stPos.nState + 20;
				END_IF
			END_IF

	16060:	stPos.sState := CONCAT(UDINT_TO_STRING(stPos.nState) ,' - Várakozás recept betöltés befejezésére');
			IF NOT fbP1RecipeManager.DONE AND NOT fbP1RecipeManager.RESET THEN
				IF NOT fbP1RecipeManager.READ_FILE.ERROR THEN
					IF bStepEnable THEN
							stPos.nState := stPos.nState + 20;			// Recept betöltés kész
					END_IF
				ELSE
					stP1PalletData.nPalletState := 1;					// Nincs recept név, viszont az SFC startolva -> le kell zárni hibával.
					stP1PalletData.nDone.4	:= TRUE;
					stP1PalletData.nErrorCode := 4104;
					eP1GapFillerCheck_Result := E_TEST_STATE.FAILED;
					stP1NcDat.MESDAT[stP1NcDat.N].RESPONSE_CODE := '4113';
					stP1NcDat.MESDAT[stP1NcDat.N].RESPONSE_DESCRIPTION := CONCAT(CONCAT('The ',arrMES_Temp[nCycle_Idx].sOP_Name),' recipe not found');
					stP1NcDat.MESDAT[stP1NcDat.N].CLIENT_DATE := fbP1MesInterface.GET_LOCAL_TIME();
					stP1NcDat.MESDAT[stP1NcDat.N].TEST_STATE := INT_TO_STRING(E_TEST_STATE.FAILED);
					stP1NcDat.MESDAT[stP1NcDat.N].TEST_STEP := INT_TO_STRING(stP1NcDat.N);
					stP1NcDat.MESDAT[stP1NcDat.N].VALUE := '0';
					stPos.nState := 95000;
				END_IF
			END_IF

	16080:	stPos.nState := 18000;


(*-----=== Normál folyamat ===-----*)
	18000:	stPos.sState := CONCAT(UDINT_TO_STRING(stPos.nState) ,' - Kiemelő munkahelyzetbe');
			fbP1Lift.bBasePosCmd := FALSE;
			fbP1Lift.bWorkPosCmd := TRUE;
			IF fbP1Lift.bWorkPosStab THEN
				IF bStepEnable THEN
					stPos.nState := stPos.nState + 20;
				END_IF
			END_IF

	18020:	stPos.sState := CONCAT(UDINT_TO_STRING(stPos.nState) ,' - Programlépés betöltése');
			fbP1AxisX.rPosition1 := LREAL_TO_REAL(stP1Recipe.Seq[i].Target.X);
			fbP1AxisX.rVelocity1 := rVelocity;
			fbP1AxisY.rPosition1 := LREAL_TO_REAL(stP1Recipe.Seq[i].Target.Y);
			fbP1AxisY.rVelocity1 := rVelocity;
			fbP1AxisZ.rPosition1 := LREAL_TO_REAL(stP1Recipe.Seq[i].Target.Z);
			fbP1AxisZ.rVelocity1 := rVelocity;
			fbP1Cam1.nProgNr := INT_TO_UINT(stP1Recipe.Seq[i].CheckingProgramId);
			IF bStepEnable THEN
					stPos.nState := stPos.nState + 20;
			END_IF
			
	18040:	stPos.sState := CONCAT(UDINT_TO_STRING(stPos.nState) ,' - X,Y,Z tengely pozícióba mozgatása');						
			fbP1AxisX.bGoPosition := TRUE;
			fbP1AxisY.bGoPosition := TRUE;
			fbP1AxisZ.bGoPosition := TRUE;
			IF fbP1AxisX.bDone AND fbP1AxisY.bDone AND fbP1AxisZ.bDone THEN
				IF bStepEnable THEN
					fbP1AxisX.bGoPosition := FALSE;
					fbP1AxisY.bGoPosition := FALSE;
					fbP1AxisZ.bGoPosition := FALSE;
					stPos.nState := stPos.nState + 20;
				END_IF
			END_IF
			
	18060:	stPos.sState := CONCAT(UDINT_TO_STRING(stPos.nState) ,' - Kamera triggerelése');						
			fbP1Cam1.bStart := TRUE;
			IF NOT fbP1Cam1.bReady AND NOT fbP1Cam1.bBusy THEN			
				IF bStepEnable THEN
					stPos.nState := stPos.nState + 20;
				END_IF
			END_IF
			
	18080:	stPos.sState := CONCAT(UDINT_TO_STRING(stPos.nState) ,' - Kiértékelés');						
			IF	fbP1Cam1.bFail THEN
					fbP1Cam1.bStart := FALSE;
					nP1ScrapCounter := nP1ScrapCounter + 1;
					stP1PalletData.nPalletState := 1;								// Fail -> Hordozólap selejt
					stP1PalletData.nDone.4	:= TRUE;
					stP1PalletData.nErrorCode := INT_TO_WORD(4121 + i);
					eP1GapFillerCheck_Result := E_TEST_STATE.FAILED;
					stP1NcDat.MESDAT[stP1NcDat.N].RESPONSE_CODE := INT_TO_STRING(4121 + i);
					stP1NcDat.MESDAT[stP1NcDat.N].RESPONSE_DESCRIPTION := CONCAT('Camera error of POS#', INT_TO_STRING(i));
					stP1NcDat.MESDAT[stP1NcDat.N].CLIENT_DATE := fbP1MesInterface.GET_LOCAL_TIME();
					stP1NcDat.MESDAT[stP1NcDat.N].TEST_STATE := INT_TO_STRING(E_TEST_STATE.FAILED);
					stP1NcDat.MESDAT[stP1NcDat.N].TEST_STEP := INT_TO_STRING(stP1NcDat.N);
					stP1NcDat.MESDAT[stP1NcDat.N].VALUE := '0';
					stPos.nState := 95000;	
			ELSE
				fbP1Cam1.bStart := FALSE;
				stPos.nState := stPos.nState + 20;
			END_IF

	18100:	stPos.sState := CONCAT(UDINT_TO_STRING(stPos.nState) ,' - Recept kész?');
			IF	stP1Recipe.Seq[i].LastPosition THEN
					IF fbP1ReceipeList.bEmpty THEN
						stPos.nState := 95000;							// A recept kész és ez volt az utolsó a listába
					ELSE
						stPos.nState := 15020;							// A recept kész de nem ez volt az utolsó a listába! -> Új recept betöltése!
					END_IF
			ELSE 
				i := i+1;												// A recept még nincs kész
				stPos.nState := 18020;
			END_IF
	
(*-----=== MES 3503 (Log NC Data) ===-----*)
	95000:	stPos.sState := CONCAT(UDINT_TO_STRING(stPos.nState) ,' - Log NC (3503)');	
			IF stP1PalletData.nPalletState = 1 AND bMesEnable THEN
				IF fbP1MesInterface.ASSY_SAVE_NCDAT(arrMES_Temp[nCycle_Idx].sDMC_Code,arrMES_Temp[nCycle_Idx].nOP_Index,stP1NcDat) THEN
					IF bStepEnable THEN
						stPos.nState := stPos.nState + 20;			// A paletta már selejt és van bent hibakód! Nincs felülírás.
					END_IF							
				END_IF
			ELSE
				IF bStepEnable THEN
					stPos.nState := stPos.nState + 20;
				END_IF
			END_IF

(*-----=== MES 3011 (Complete SFC) ===-----*)
	95020:	stPos.sState := CONCAT(UDINT_TO_STRING(stPos.nState) ,' - Complete SFC (3011)');
			IF bMesEnable THEN	
				IF fbP1MesInterface.COMPLETE_SFC(arrMES_Temp[nCycle_Idx].sDMC_Code, arrMES_Temp[nCycle_Idx].nOP_Index, eP1GapFillerCheck_Result) THEN
					IF stP1MesResp.RESP_CODE='0' THEN
						stPos.nState := stPos.nState + 20;
					ELSE
						stP1PalletData.nPalletState := 1;			// A MES-be aktív marad nem tudom selejtezni! Csak a hordozót selejtezem
						stP1PalletData.nErrorCode := 4114;
						stPos.nState := stPos.nState + 20;
					END_IF
				END_IF
			ELSE
				stPos.nState := stPos.nState + 20;
			END_IF


	95040:	stPos.sState := CONCAT(UDINT_TO_STRING(stPos.nState) ,' - Folyamat ellenőrzése');
			IF stP1PalletData.nPalletState = 1 OR nCycle_Idx >= 2 THEN
				IF bStepEnable THEN						// Selejt vagy kész a folyamat -> Lejelentés
					stP1PalletData.nDone.4 := TRUE;
					stPos.nState := stPos.nState + 20;
				END_IF
			ELSE
				IF bStepEnable THEN
					nCycle_Idx := nCycle_Idx + 1;		// Jó termék és még nincs kész a folyamat -> Mehet a köv. folyamat
					IF bMesEnable THEN
						stPos.nState := 15000;
					ELSE
						stPos.nState := 16000;
					END_IF
				END_IF
			END_IF
			
	95060:		
			stPos.nState := 96000;

	(*-----=== Hordozólap adatok feltöltése ST10-be ===-----*)
	96000:	stPos.sState := CONCAT(UDINT_TO_STRING(stPos.nState) ,' - Paletta adatok feltöltése');
			fbP1PalletDataExchange.nIndex := fbP1RFID.nTAGData;
			IF bStepEnable THEN
				fbP1PalletDataExchange.eCommand := Write;
				stPos.nState := stPos.nState + 20;
			END_IF
			
	(*-----=== Hordozólap adatok feltöltése ST10-be ===-----*)
	96020:	stPos.sState := CONCAT(UDINT_TO_STRING(stPos.nState) ,' - Paletta adatok feltöltése');
			IF fbP1PalletDataExchange.bDone AND NOT fbP1PalletDataExchange.bError THEN
				IF bStepEnable THEN
					fbP1PalletDataExchange.eCommand := NoCmd;
					stPos.nState := stPos.nState + 20;
				END_IF
			END_IF

	96040:	stPos.sState := CONCAT(UDINT_TO_STRING(stPos.nState) ,' - X,Y tengely pozícióba mozgatása');
			fbP1AxisX.rPosition1 := 0;
			fbP1AxisX.rVelocity1 := rVelocity;
			fbP1AxisY.rPosition1 := 0;
			fbP1AxisY.rVelocity1 := rVelocity;					
			fbP1AxisZ.rPosition1 := 0;
			fbP1AxisZ.rVelocity1 := rVelocity;					
			fbP1AxisX.bGoPosition := TRUE;
			fbP1AxisY.bGoPosition := TRUE;
			fbP1AxisZ.bGoPosition := TRUE;
			IF fbP1AxisX.bDone AND fbP1AxisY.bDone AND fbP1AxisZ.bDone THEN
				IF bStepEnable THEN
					fbP1AxisX.bGoPosition := FALSE;
					fbP1AxisY.bGoPosition := FALSE;
					fbP1AxisZ.bGoPosition := FALSE;
					stPos.nState := stPos.nState + 20;
				END_IF
			END_IF		
	
	96060:	stPos.sState := CONCAT(UDINT_TO_STRING(stPos.nState) ,' - Kiemelő alaphelyzetbe');
			fbP1Lift.bBasePosCmd := TRUE;
			fbP1Lift.bWorkPosCmd := FALSE;
			IF fbP1Lift.bBasePosStab THEN
				IF bStepEnable THEN
					i:=0;
					stPos.nState := stPos.nState + 20;	
				END_IF
			END_IF		

	96080:	stPos.sState := CONCAT(UDINT_TO_STRING(stPos.nState) ,' - Ismétlődő hibák ellenőrzése');
			IF NOT bP1ScrapRepeatError THEN
				stPos.nState := 100000;
			END_IF
{endregion}
			
(*-----=== Automata ciklus befejezése ===-----*)
	100000:	stPos.sState := CONCAT(UDINT_TO_STRING(stPos.nState) ,' - Várakozás hordozólap elengedésre');
			IF NOT fbP1Stopper.bPalletAtStopper THEN
				IF bStepEnable THEN
					i:=0;
					stPos.nState := stPos.nState + 20;
				END_IF
			END_IF		

	100020:
			stPos.nState := 10000;	
			
(* Kézi üzem *********************************************************************)
	150000:	stPos.sState := CONCAT(UDINT_TO_STRING(stPos.nState) ,' - Kézi üzem');
			IF NOT bManualMode THEN
				stPos.nState := 0;
			ELSE
				;
			END_IF
			
	(* Hibakezelés *********************************************************************)
	200000:	stPos.sState := CONCAT(UDINT_TO_STRING(stPos.nState) ,CONCAT(' - Hiba, ebből az állapotból: ' ,stPos.sState));
			fbP1PalletDataExchange.eCommand := NoCmd;
			stPos.bError := TRUE;
			stPos.nState := stPos.nState + 20;

	(* Hibakezelés *********************************************************************)
	200020:	IF bAckP THEN
				CASE stPos.nStateLast OF
					(* Alaphelyzet felvétel folyamán *)
					0..9999:	stPos.nState := 0;
				ELSE 			stPos.nState := 0;
				END_CASE
				stPos.bError := FALSE;
			END_IF
ELSE
	stPos.sState := CONCAT(UDINT_TO_STRING(stPos.nState) ,' - Nem használt állapot');
END_CASE

ACTION Camera:
fbP1Cam1(
	sName:= 'CAM1 Basler acA4600-7gc', 
	bEn:= TRUE, 
	bEHA:= TRUE, 
	bAck:= bAckP, 
	timConnection:= T#1500MS, 
	timReady:= T#1500MS, 
	timProgChange:= T#1500MS, 
	timProgRun:= T#5S, 
	stCAM_IN:= stCam1_IN,
	stComErrEvent:= TC_EVENTS.MyEvent.fbP1Cam1Com,
	stReadyErrEvent:= TC_EVENTS.MyEvent.fbP1Cam1Ready,
	stProgErrEvent:= TC_EVENTS.MyEvent.fbP1Cam1Prog,
	stRunErrEvent:= TC_EVENTS.MyEvent.fbP1Cam1Run, 
	stCAM_OUT=> stCam1_OUT);
END_ACTION

ACTION DataExchange:
fbP1PalletDataExchange(
	stPalletData:= stP1PalletData, 
	sName:= 'P1 Camera pos.', 
	bAck:= bAckP, 
	sAMSNetId:= sST10_NetId, 
	stEventEntry:= TC_EVENTS.MyEvent.fbP1PalletDataExchange);
END_ACTION

ACTION Diag:
fbP1FullCycleTime(
	bPalletSensor:= fbP1Stopper.i_bPalettSensor,
	timTimeMax:= T#200S,
	nCurrentCycleTime=> ,
	arrCycleTimes=> );
END_ACTION

ACTION MES:
fbP1MesInterface(
	HOST:= '127.0.0.1', 
	PORT:= 5500, 
	ENABLE:= TRUE, 
	RESET:= fbP1MesInterface.ERROR, 
	STX:= , 
	ETX:= , 
	RESP:= stP1MesResp, 
	TEST_ADAPTER:= '0', 
	ADAPTER_ID:= '1', 
	BUSY=> , 
	READY=> , 
	DONE=> , 
	ERROR=> , 
	ERROR_ID=> );
END_ACTION

ACTION Pneu:
fbP1Lift(
	sName:= 'Z4.4', 
	sBasePosSensor:= 'S4131', 
	sWorkPosSensor:= 'S4132', 
	bEn:= i_bDoorOK, 
	bEHA:= bGlobalEHA, 
	bDisableManualCmd:= NOT bManualMode, 
	bAck:= bAckP, 
	timBasePos:= , 
	timWorkPos:= ,
	stBasePosEvent:= TC_Events.MyEvent.fbP1LiftBPE, 
	stWorkPosEvent:= TC_Events.MyEvent.fbP1LiftWPE);
END_ACTION

ACTION Recipe:
fbP1RecipeManager(
	sDef:= 'Vision', 
	sExt:= 'tcdata', 
	sFolderPath:= 'C:\TwinCAT\Tc_Data', 
	sKey:= 'Data', 
	pData:= ADR(stP1Recipe), 
	nData:= SIZEOF(stP1Recipe), 
	RESET:= , 
	READY=> , 
	BUSY=> , 
	DONE=> , 
	ERROR=> , 
	ERROR_ID=> , 
	TIME_STAMP=> , 
	RECIPE_LIST=> arrP1RecipeNames, 
	RECIPE_CNT=> );
	
IF	bP1RecipeLoad AND
	NOT bP1RecipeSave AND
	NOT bP1RecipeRefresh AND
	NOT fbP1RecipeManager.RESET AND
	NOT fbP1RecipeManager.DONE THEN
			fbP1RecipeManager.Load(NAME:= sP1RecipeName);
END_IF

IF	NOT bP1RecipeLoad AND
	bP1RecipeSave AND
	NOT bP1RecipeRefresh AND
	NOT fbP1RecipeManager.RESET AND
	NOT fbP1RecipeManager.DONE THEN
			fbP1RecipeManager.Save(NAME:= sP1RecipeName);
END_IF

IF	NOT bP1RecipeLoad AND
	NOT bP1RecipeSave AND
	bP1RecipeRefresh AND
	NOT fbP1RecipeManager.RESET AND
	NOT fbP1RecipeManager.DONE THEN
			fbP1RecipeManager.RefreshNameList();
END_IF

IF	NOT bP1RecipeLoad AND
	NOT bP1RecipeSave AND
	NOT bP1RecipeRefresh AND
	NOT fbP1RecipeManager.RESET AND
	fbP1RecipeManager.DONE THEN
			fbP1RecipeManager.RESET := TRUE;
END_IF

IF	fbP1RecipeManager.RESET AND
	NOT fbP1RecipeManager.DONE THEN
			fbP1RecipeManager.RESET := FALSE;
END_IF
END_ACTION

ACTION RFID:
fbP1RFID(sName:= 'P1 RFID');
END_ACTION

ACTION Servo:
fbP1AxisX.lrNegLimit := 0;
fbP1AxisX.lrPosLimit := 390;
fbP1AxisX.bEnableNegative := TRUE;
fbP1AxisX.bEnablePositive := TRUE;

fbP1AxisX(
	sName:= 'Axis X', 
	bEMYOK:= i_bDoorOK AND NOT i_bAX5805ErrorX, 
	bErrorAck:= bAckP, 
	bDisableManualCmd:= NOT bManualMode, 
	bBufferedMove:= FALSE,
	rVelocityJog := 10, 
	stAxisEvent:= TC_EVENTS.MyEvent.fbP1AxisX
);

fbP1AxisY.lrNegLimit := 0;
fbP1AxisY.lrPosLimit := 290;
fbP1AxisY.bEnableNegative := TRUE;
fbP1AxisY.bEnablePositive := TRUE;

fbP1AxisY(
	sName:= 'Axis Y', 
	bEMYOK:= i_bDoorOK AND NOT i_bAX5805ErrorY, 
	bErrorAck:= bAckP, 
	bDisableManualCmd:= NOT bManualMode, 
	bBufferedMove:= FALSE, 
	rVelocityJog := 10, 
	stAxisEvent:= TC_EVENTS.MyEvent.fbP1AxisY
);

fbP1AxisZ.lrNegLimit := 0;
fbP1AxisZ.lrPosLimit := 100;
fbP1AxisZ.bEnableNegative := TRUE;
fbP1AxisZ.bEnablePositive := TRUE;

fbP1AxisZ(
	sName:= 'Axis Z', 
	bEMYOK:= i_bDoorOK AND NOT i_bAX5805ErrorZ, 
	bErrorAck:= bAckP, 
	bDisableManualCmd:= NOT bManualMode, 
	bBufferedMove:= FALSE, 
	rVelocityJog := 10, 
	stAxisEvent:= TC_EVENTS.MyEvent.fbP1AxisZ
);
END_ACTION

END_PROGRAM

// ---- POUs/P2_Robot.TcPOU
PROGRAM P2_Robot
VAR
	stPos					:ST_PosData;
	tCycleTime				:TON;
	bInProcess				:BOOL := FALSE;
	bPcbaScrap				:BOOL := FALSE;
END_VAR

(*Időzítők***************************************************)
IF (stPos.nState>10000) AND (stPos.nState<100000) AND NOT tCycleTime.Q THEN
	stPos.nCycleTime := TIME_TO_REAL(tCycleTime.ET)/1000;
END_IF
tCycleTime(IN:= (stPos.nState>10000) AND (stPos.nState<150000), PT:= T#200S);							// A palettára várakozás nincs beszámolva
(*Triggerek**************************************************)

(*Vész rendszer**********************************************)
IF	(NOT (i_bEmyOK AND fbDoor.bDoorsLocked) AND stPos.nState > 0) OR									// Nincs vészkör, vagy
	(NOT i_bDoorOK AND (stPos.nState>=60 AND stPos.nState<=1000)) OR									// alaphelyzetfelvétel közbe megszűnik az ajtókör vagy
	(NOT i_bDoorOK AND (stPos.nState>=10060 AND stPos.nState<=100060)) THEN							// folyamat közbe megszűnik az ajtókör 
		stPos.nState := 0;
END_IF;

(*Hibakezelés************************************************)
IF stPos.nState > 0 AND stPos.nState < 150000 THEN
	stPos.nStateLast := stPos.nState;
	IF	fbP2Lift.bError OR
		fbP2PalletDataExchange.bError OR
		fbP2KRC4.bError OR
		(NOT fbP2KRC4.bReady AND stPos.nState >= 10000 AND stPos.nState < 150000) OR
		stPos.bError THEN
			stPos.nState := 200000;
	END_IF
END_IF

(*Engedélyek *************************************************)
IF stPos.nState <= 10000
	OR stPos.nState = 150000
	OR stPos.nState = 100000
	OR stPos.nState >= 200000
THEN
	stPos.bManualModeEnable := TRUE;
ELSE
	stPos.bManualModeEnable := FALSE;
END_IF

IF stPos.nState = 0
	OR stPos.nState = 10000
	OR stPos.nState = 100000
	OR stPos.nState = 150000
	OR stPos.nState >= 200000
THEN
	stPos.bDoorOpenEnable := TRUE;
ELSE
	stPos.bDoorOpenEnable := FALSE;
END_IF

(*Kézi üzem *************************************************)
IF	bManualMode OR
	NOT fbP2KRC4.RobotIn.Status.bExt THEN						// A pendantról is manuálba lehet küldeni.
		stPos.nState := 150000;
END_IF

(*Automata üzem *********************************************)
CASE stPos.nState OF
{region "Init process"}
	0:		stPos.sState := CONCAT(UDINT_TO_STRING(stPos.nState) ,' - Vészkör vagy ajtókör bontva - Működtetések törlése');
			fbP2Lift.bBasePosCmd := TRUE;
			fbP2Lift.bWorkPosCmd := FALSE;
			fbP2KRC4.bAutoCycle := FALSE;
			fbP2KRC4.bExecuteProg := FALSE;
			fbP2KRC4.nProgNr := 0;
			fbP2PalletDataExchange.eCommand := NoCmd;
			stPos.bError := FALSE;
			stPos.nErrorCode := 0;
			IF i_bDoorOK THEN
				IF bStepEnable THEN
					stPos.nState := stPos.nState + 20;
				END_IF
			END_IF
			
	20:		stPos.sState := CONCAT(UDINT_TO_STRING(stPos.nState) ,' - Alaphelyzetfelvétel - Kiemelő ellenőrzése');
			IF fbP2Lift.i_bBasePos THEN
				IF bStepEnable THEN								// A kiemelő alaphelyzetbe volt akkor nincs kiemelés
					stPos.nState := 100;
				END_IF
			ELSE
				IF bStepEnable THEN								// A paletta már ki volt emelve -> Lehet hogy a robot még a PCB alatt van
					stPos.nState := 200;							// ezért ki kell emelni a palettát különben valami törni fog !
				END_IF
			END_IF


	100:	stPos.sState := CONCAT(UDINT_TO_STRING(stPos.nState) ,' - Alaphelyzetfelvétel - Kiemelő alaphelyzetbe');
			fbP2Lift.bBasePosCmd := TRUE;
			fbP2Lift.bWorkPosCmd := FALSE;
			IF fbP2Lift.bBasePosStab THEN
				IF bStepEnable THEN
					stPos.nState := 300;
				END_IF
			END_IF

	200:	stPos.sState := CONCAT(UDINT_TO_STRING(stPos.nState) ,' - Alaphelyzetfelvétel - Kiemelő munkahelyzetbe');
			fbP2Lift.bBasePosCmd := FALSE;
			fbP2Lift.bWorkPosCmd := TRUE;
			IF fbP2Lift.bWorkPosStab THEN
				IF bStepEnable THEN
					stPos.nState := 300;
				END_IF
			END_IF

	300:	stPos.sState := CONCAT(UDINT_TO_STRING(stPos.nState) ,' - Alaphelyzetfelvétel - Várakozás robot zóna engedélyre');
			IF fbP2KRC4.bZoneEnable THEN
				IF bStepEnable THEN
					stPos.nState := 400;
				END_IF
			END_IF

	400:	stPos.sState := CONCAT(UDINT_TO_STRING(stPos.nState) ,' - Alaphelyzetfelvétel - Várakozás robot alaphelyzetfelvételre');
			IF fbP2KRC4.bReady AND NOT fbP2KRC4.bBusy THEN
				IF bStepEnable THEN
					stPos.nState := stPos.nState + 20;
				END_IF
			END_IF			

	420:	stPos.sState := CONCAT(UDINT_TO_STRING(stPos.nState) ,' - Alaphelyzetfelvétel - Kiemelő alaphelyzetbe');
			fbP2Lift.bBasePosCmd := TRUE;
			fbP2Lift.bWorkPosCmd := FALSE;
			IF fbP2Lift.bBasePosStab THEN
				IF bStepEnable THEN
					stPos.nState := stPos.nState + 20;
				END_IF
			END_IF
			
	440:	stPos.sState := CONCAT(UDINT_TO_STRING(stPos.nState) ,' - Alaphelyzetfelvétel - Robot ellenőrzése');
			IF	fbP2KRC4.RobotIn.Status.bVacuumOutStat OR				// Robot vákuum bekapcsolva
				fbP2KRC4.RobotIn.Status.bVacuumInStat OR				// Robot vákuum visszajelzés
				fbP2KRC4.RobotIn.Status.bProdSensor THEN				// Darabérzékelő visszajelzés
					;															// A robotnál alkatrész van -> El kell tőle venni! => LINE STOP!!!
			ELSE
					stPos.nState := stPos.nState + 20;	 
			END_IF

	460:	stPos.sState := CONCAT(UDINT_TO_STRING(stPos.nState) ,' - Alaphelyzetfelvétel - Megkezdett folyamat ellenőrzése');
			IF bInProcess THEN
				stP2PalletData.nPalletState := 1;
				stP2PalletData.nErrorCode := 4209;
				stP2NcDat.N := 1;
				eP2Assy_Auto2_Result := E_TEST_STATE.FAILED;
				stP2NcDat.MESDAT[stP2NcDat.N].RESPONSE_CODE := '4209';
				stP2NcDat.MESDAT[stP2NcDat.N].RESPONSE_DESCRIPTION := 'Process error ';
				stP2NcDat.MESDAT[stP2NcDat.N].CLIENT_DATE := fbP2MesInterface.GET_LOCAL_TIME();
				stP2NcDat.MESDAT[stP2NcDat.N].TEST_STATE := INT_TO_STRING(E_TEST_STATE.FAILED);
				stP2NcDat.MESDAT[stP2NcDat.N].TEST_STEP := INT_TO_STRING(stP2NcDat.N);
				stP2NcDat.MESDAT[stP2NcDat.N].VALUE := '0';
				stPos.nState := stPos.nState + 20;
			ELSE
				stPos.nState := 600;
			END_IF

	 
//	480:	stP2.nState := 95000;
		 
			  
	480:	stPos.sState := CONCAT(UDINT_TO_STRING(stPos.nState) ,' - Alaphelyzetfelvétel - PCBA selejtezése');
		 	IF bPcbaScrap THEN
				IF fbP2MesInterface.SCRAP_SFC(stP2PalletData.sPCBACode, nP2Assy_Auto2_Index) THEN
					bPcbaScrap := false;
					stPos.nState := 19000;
				END_IF
			ELSE
				stPos.nState := 95000;
			END_IF	 
		  		
	600:	stPos.nState := 10000;
{endregion}			
			
(* Alaphelyzet *********************************************************************)
	10000:	stPos.sState := CONCAT(UDINT_TO_STRING(stPos.nState) ,' - Alaphelyzet, termékre vár');
			IF fbP2RFID.bTagPresent AND fbP2Stopper.bPalletAtStopper AND NOT bP2ScrapRepeatError  THEN
				IF bStepEnable THEN
					stPos.nState := stPos.nState + 20;	
				END_IF
			END_IF	

	(*-----=== Hordozólap adatok lekérdezése ST10-től ===-----*)
	10020:	stPos.sState := CONCAT(UDINT_TO_STRING(stPos.nState) ,' - Paletta adatok lekérdezése');
			fbP2PalletDataExchange.nIndex := fbP2RFID.nTAGData;
			IF bStepEnable THEN
				fbP2PalletDataExchange.eCommand := Read;
				stPos.nState := stPos.nState + 20;
			END_IF
			
	(*-----=== Hordozólap adatok lekérdezése ST10-től ===-----*)
	10040:	stPos.sState := CONCAT(UDINT_TO_STRING(stPos.nState) ,' - Paletta adatok lekérdezése');
			IF fbP2PalletDataExchange.bDone AND NOT fbP2PalletDataExchange.bError THEN
				IF bStepEnable THEN
					fbP2PalletDataExchange.eCommand := NoCmd;
					stPos.nState := stPos.nState + 20;
				END_IF
			END_IF

	(*-----=== Hordozólap adatok kiértékelése ===-----*)
	10060:	stPos.sState := CONCAT(UDINT_TO_STRING(stPos.nState) ,' - Paletta adatok lekérdezése');
			IF		stP2PalletData.nPalletState = 2 AND			// OK termék a palettán
					stP2PalletData.nDone.4 AND					// Kamerás ell. kész
					NOT stP2PalletData.nDone.5 THEN				// Összeszerelés még nincs kész
						IF bStepEnable THEN						// Mehet a kiemelés -> Normál folyamat
							stPos.nState := stPos.nState + 20;
						END_IF
			ELSIF	stP2PalletData.nPalletState = 42 THEN		// Teszt hordozólap a kamerához
						IF bStepEnable THEN						// Még nincs funkció -> Tovább engedés
							stPos.nState := 96000;
						END_IF
			ELSIF	stP2PalletData.nPalletState = 2 AND			// OK termék a palettán
					NOT stP2PalletData.nDone.4 THEN				// Kamerás ell. nincs kész !
						IF bStepEnable THEN						// Átemelt hordozólap!?!? -> Selejtezés
							stP2PalletData.nPalletState := 1;
							stP2PalletData.nDone.5 := TRUE;	
							stP2PalletData.nErrorCode := 4200;
							stPos.nState := 96000;
						END_IF
			ELSIF	stP2PalletData.nPalletState = 1 THEN		// Selejt termék a palettán
						IF bStepEnable THEN						// Nincs kiemelés -> Tovább engedés
							stPos.nState := 96060;
						END_IF
			ELSIF	stP2PalletData.nPalletState = 0 THEN		// Üres paletta
						IF bStepEnable THEN						// Nincs kiemelés -> Tovább engedés
							stPos.nState := 96060;
						END_IF
			ELSE												// Nincs teendő, más állomásnak szánt hordozólap
						IF bStepEnable THEN						// Nincs kiemelés -> Tovább engedés
							stPos.nState := 96060;
						END_IF			
			END_IF


	(*-----=== Alkatrészek ellenőrzése a palettán ===-----*)
	10080:	stPos.sState := CONCAT(UDINT_TO_STRING(stPos.nState) ,' - Alkatrészek ellenőrzése a palettán');
			IF	i_bP2DutSensor1 AND
				i_bP2DutSensor2 AND
				i_bP2DutSensor3 AND
				NOT i_bP2PalletSensor THEN
					IF bStepEnable THEN							// Minden a helyén mehet az összeszerelés
						stPos.nState := stPos.nState + 20;
					END_IF
			ELSE
					IF bStepEnable THEN							// Hiányzó alkatrészek -> Nem lehet összeépíteni -> selejtezés
						stP2PalletData.nPalletState := 1;		// Paletta selejtre jelentése
						stP2PalletData.nDone.5 := TRUE;			// Állomás készre jelentése
						stP2PalletData.nErrorCode := 4201;		// Hibakód beírása
 						stPos.nState := 96000;					// Paletta adatok tárolása.
					END_IF				
			END_IF

	(*-----=== MES engedély ellenőrzése ===-----*)
	10100:	stPos.sState := CONCAT(UDINT_TO_STRING(stPos.nState) ,' - MES Engedély ellenőrzése');
			IF bMesEnable THEN
				IF bStepEnable THEN
					stPos.nState := 15000;
				END_IF
			ELSE
				IF bStepEnable THEN
					stPos.nState := 16000;
				END_IF				
			END_IF

	(*-----=== MES 3010 (Start SFC) ===-----*)	
	15000:	stPos.sState := CONCAT(UDINT_TO_STRING(stPos.nState) ,' - Start SFC (3010)');	
			IF bMesEnable THEN
				IF fbP2MesInterface.START_SFC(stP2PalletData.sMRTCode, nP2Assy_Auto2_Index) THEN
					IF stP2MesResp.RESP_CODE='0' THEN
						IF bStepEnable THEN
							bInProcess := TRUE;
							stPos.nState := stPos.nState + 20;
						END_IF
					ELSE
						IF bStepEnable THEN
							stP2PalletData.nPalletState := 1;		// Paletta selejtre jelentése
							stP2PalletData.nDone.5 := TRUE;			// Állomás készre jelentése
							stP2PalletData.nErrorCode := 4202;		// Hibakód beírása
							stPos.nState := 96000;					// Paletta adatok tárolása.
						END_IF
					END_IF
				END_IF
			ELSE
				IF bStepEnable THEN
					bInProcess := TRUE;
					stPos.nState := stPos.nState + 20;
				END_IF	
			END_IF

	15020:	stPos.nState := 16000;	
		
(*-----=== Recept betöltés ===-----*)
	16000:
			IF bStepEnable THEN
				stPos.nState := 18000;
			END_IF	

(*-----=== Normál folyamat ===-----*)
	18000:	stPos.sState := CONCAT(UDINT_TO_STRING(stPos.nState) ,' - Kiemelő munkahelyzetbe');
			fbP2Lift.bBasePosCmd := FALSE;
			fbP2Lift.bWorkPosCmd := TRUE;
			IF fbP2Lift.bWorkPosStab THEN
				IF bStepEnable THEN
					stPos.nState := stPos.nState + 20;
				END_IF
			END_IF

	18020:	stPos.sState := CONCAT(UDINT_TO_STRING(stPos.nState) ,' - PCBA felvétele a hordozólapról');
			fbP2KRC4.nProgNr := 10;
			fbP2KRC4.bExecuteProg := TRUE;
			IF fbP2KRC4.bDone THEN
				fbP2KRC4.bExecuteProg := FALSE;
				IF bStepEnable THEN
					stPos.nState := stPos.nState + 20;
				END_IF
			END_IF			
			
	18040:	stPos.sState := CONCAT(UDINT_TO_STRING(stPos.nState) ,' - PCBA behelyezése');
			fbP2KRC4.nProgNr := 11;
			fbP2KRC4.bExecuteProg := TRUE;
			IF fbP2KRC4.bDone THEN
				fbP2KRC4.bExecuteProg := FALSE;
				IF bStepEnable THEN
					stPos.nState := stPos.nState + 20;
				END_IF
			END_IF			
						
	18060:	stPos.sState := CONCAT(UDINT_TO_STRING(stPos.nState) ,' - Cover felvétele a hordozólapról');
			fbP2KRC4.nProgNr := 12;
			fbP2KRC4.bExecuteProg := TRUE;
			IF fbP2KRC4.bDone THEN
				fbP2KRC4.bExecuteProg := FALSE;
				IF bStepEnable THEN
					stPos.nState := stPos.nState + 20;
				END_IF
			END_IF			

(*												//	Ciklusidő gyorsítás miatt Interlock bit figyelése a Done bit helyett 2021.03.25 ZZs		
	18080:	stP2.sState := CONCAT(UDINT_TO_STRING(stP2.nState) ,' - Cover behelyezése');
			fbP2KRC4.nProgNr := 13;
			fbP2KRC4.bExecuteProg := TRUE;
			IF fbP2KRC4.bDone THEN
				fbP2KRC4.bExecuteProg := FALSE;
				IF bStepEnable THEN
					stP2PalletData.nDone.5 := TRUE;
					stP2.nState := stP2.nState + 20;
				END_IF
			END_IF					
*)
	18080:	stPos.sState := CONCAT(UDINT_TO_STRING(stPos.nState) ,' - Cover behelyezése');
			fbP2KRC4.nProgNr := 13;
			fbP2KRC4.bExecuteProg := TRUE;
			IF fbP2KRC4.RobotIn.Status.bIntMoveInPalettZone THEN
				IF bStepEnable THEN
					stPos.nState := stPos.nState + 20;
				END_IF
			END_IF					

	18100:	stPos.sState := CONCAT(UDINT_TO_STRING(stPos.nState) ,' - Várakozás Cover behelyezésére');			
			IF NOT fbP2KRC4.RobotIn.Status.bIntMoveInPalettZone THEN
				IF bStepEnable THEN
					stP2PalletData.nDone.5 := TRUE;
					stPos.nState := stPos.nState + 20;
				END_IF
			END_IF					

	18120:
(*
Inventory sorrend
0:	MRT
1:	Carrier
2:	Cover
3:	PCBA
4:	Fan
*)
			stP2MrtInventoryList.LIST[0] := stP2PalletData.stInventoryList.LIST[3];			// PCBA
			stP2MrtInventoryList.LIST[1] := stP2PalletData.stInventoryList.LIST[2];			// Cover
			stP2MrtInventoryList.LIST[2] := stP2PalletData.stInventoryList.LIST[4];			// FAN
			stPos.nState := stPos.nState + 20;
			
(*-----=== MES  (Assembly by inventory 2138) ===-----*)
	18140:	stPos.sState := CONCAT(UDINT_TO_STRING(stPos.nState) ,' - Assemble inventory (2138)');
			IF bMesEnable THEN	
				IF fbP2MesInterface.ASSEMBLE_BY_INVENTORY_LIST(stP2PalletData.sMRTCode, nP2Assy_Auto2_Index, stP2MrtInventoryList) THEN
					IF stP2MesResp.RESP_CODE='0' THEN
						eP2Assy_Auto2_Result:=E_TEST_STATE.PASSED;
					ELSE
						stP2PalletData.nPalletState := 1;				// Paletta selejtre jelentése
						stP2PalletData.nDone.5 := TRUE;					// Állomás készre jelentése
						stP2PalletData.nErrorCode := 4210;				// Hibakód beírása
						stP2NcDat.N := 1;
						eP2Assy_Auto2_Result := E_TEST_STATE.FAILED;
						stP2NcDat.MESDAT[stP2NcDat.N].RESPONSE_CODE := '4210';
						stP2NcDat.MESDAT[stP2NcDat.N].RESPONSE_DESCRIPTION := 'Process error ';
						stP2NcDat.MESDAT[stP2NcDat.N].CLIENT_DATE := fbP2MesInterface.GET_LOCAL_TIME();
						stP2NcDat.MESDAT[stP2NcDat.N].TEST_STATE := INT_TO_STRING(E_TEST_STATE.FAILED);
						stP2NcDat.MESDAT[stP2NcDat.N].TEST_STEP := INT_TO_STRING(stP2NcDat.N);
						stP2NcDat.MESDAT[stP2NcDat.N].VALUE := '0';
					END_IF
					IF bStepEnable THEN
						stPos.nState := stPos.nState + 20;
					END_IF
				END_IF
			ELSE
				IF bStepEnable THEN
					stPos.nState := stPos.nState + 20;
				END_IF
			END_IF

	18160:	stPos.nState := 95000;

(*-----=== MES 503 (Log Nc) ===-----*)
	95000:	stPos.sState := CONCAT(UDINT_TO_STRING(stPos.nState) ,' - Log Nc data (503)  MRT');
			IF stP2PalletData.nPalletState = 1 AND bMesEnable THEN	
				IF fbP2MesInterface.ASSY_SAVE_NCDAT(stP2PalletData.sMRTCode,nP2Assy_Auto2_Index,stP2NcDat) THEN
						IF bStepEnable THEN
							stPos.nState := stPos.nState + 20;
						END_IF							
				END_IF
			ELSE
				stPos.nState := stPos.nState + 20;	
			END_IF

(*-----=== MES 3011 (Complete SFC) ===-----*)
	95020:	stPos.sState := CONCAT(UDINT_TO_STRING(stPos.nState) ,' - Complete SFC (3011)');	
			IF bMesEnable THEN
				IF fbP2MesInterface.COMPLETE_SFC(stP2PalletData.sMRTCode, nP2Assy_Auto2_Index, eP2Assy_Auto2_Result) THEN
					IF stP2MesResp.RESP_CODE='0' THEN
						IF bStepEnable THEN
								stPos.nState := 96000;
						END_IF
					ELSE
						IF bStepEnable THEN
								stP2PalletData.nPalletState := 1;				// Paletta selejtre jelentése
								stP2PalletData.nDone.5 := TRUE;					// Állomás készre jelentése
								stP2PalletData.nErrorCode := 4205;				// Hibakód beírása
								stPos.nState := 96000;
						END_IF
					END_IF
				END_IF
			ELSE
				IF bStepEnable THEN
						stPos.nState := 96000;
				END_IF
			END_IF

	(*-----=== Hordozólap adatok feltöltése ST10-be ===-----*)
	96000:	stPos.sState := CONCAT(UDINT_TO_STRING(stPos.nState) ,' - Paletta adatok feltöltése');
			fbP2PalletDataExchange.nIndex := fbP2RFID.nTAGData;
			IF bStepEnable THEN
				fbP2PalletDataExchange.eCommand := Write;
				stPos.nState := stPos.nState + 20;
			END_IF
			
	(*-----=== Hordozólap adatok feltöltése ST10-be ===-----*)
	96020:	stPos.sState := CONCAT(UDINT_TO_STRING(stPos.nState) ,' - Paletta adatok feltöltése');
			IF fbP2PalletDataExchange.bDone AND NOT fbP2PalletDataExchange.bError THEN
				IF bStepEnable THEN
					fbP2PalletDataExchange.eCommand := NoCmd;
					stPos.nState := stPos.nState + 20;
				END_IF
			END_IF

	96040:	stPos.nState := 96060;	
	
	(*-----=== Normál folyamat kész ===-----*)		
	96060:	stPos.sState := CONCAT(UDINT_TO_STRING(stPos.nState) ,' - Kiemelő alaphelyzetbe');
			bInProcess := FALSE;
			fbP2Lift.bBasePosCmd := TRUE;
			fbP2Lift.bWorkPosCmd := FALSE;
			IF fbP2Lift.bBasePosStab THEN
				IF bStepEnable THEN
					stPos.nState := stPos.nState + 20;
				END_IF
			END_IF		

	96080:	stPos.sState := CONCAT(UDINT_TO_STRING(stPos.nState) ,' - Ismétlődő hibák ellenőrzése');
			IF NOT bP2ScrapRepeatError THEN
				stPos.nState := 100000;
			END_IF

(*-----=== Automata ciklus befejezése ===-----*)
	100000:	stPos.sState := CONCAT(UDINT_TO_STRING(stPos.nState) ,' - Várakozás hordozólap elengedésre');
			IF NOT fbP2Stopper.bPalletAtStopper THEN
				IF bStepEnable THEN
					stPos.nState := stPos.nState + 20;
				END_IF
			END_IF		

	100020:	stPos.sState := CONCAT(UDINT_TO_STRING(stPos.nState) ,' - Robot vezérlő bitek törlése');
			IF fbP2KRC4.bDone OR NOT fbP2KRC4.bExecuteProg THEN
				fbP2KRC4.bExecuteProg := FALSE;
				IF bStepEnable THEN
					stPos.nState := 10000;
				END_IF
			END_IF	

			
(* Kézi üzem *********************************************************************)
	150000:	stPos.sState := CONCAT(UDINT_TO_STRING(stPos.nState) ,' - Kézi üzem');
			IF 	NOT bManualMode AND
				fbP2KRC4.RobotIn.Status.bExt THEN					// A robotnak is external-ba kell lennie!
					stPos.nState := 0;
			ELSE
				;
			END_IF
			
	(* Hibakezelés *********************************************************************)
	200000:	stPos.sState := CONCAT(UDINT_TO_STRING(stPos.nState) ,CONCAT(' - Hiba, ebből az állapotból: ' ,stPos.sState));
			fbP2PalletDataExchange.eCommand := NoCmd;
			stPos.bError := TRUE;
			stPos.nState := stPos.nState + 20;

	(* Hibakezelés *********************************************************************)
	200020:	IF bAckP THEN
				CASE stPos.nStateLast OF
					(* Alaphelyzet felvétel folyamán *)
					0..9999:	stPos.nState := 0;
				ELSE 			stPos.nState := 0;
				END_CASE
				stPos.bError := FALSE;
			END_IF
ELSE
	stPos.sState := CONCAT(UDINT_TO_STRING(stPos.nState) ,' - Nem használt állapot');
END_CASE

ACTION DataExchange:
fbP2PalletDataExchange(
	stPalletData:= stP2PalletData, 
	sName:= 'P2 Robot pos.', 
	bAck:= bAckP, 
	sAMSNetId:= sST10_NetId, 
	stEventEntry:= TC_EVENTS.MyEvent.fbP2PalletDataExchange);
END_ACTION

ACTION Diag:
fbP2FullCycleTime(
	bPalletSensor:= fbP2Stopper.i_bPalettSensor,
	timTimeMax:= T#200S,
	nCurrentCycleTime=> ,
	arrCycleTimes=> );
END_ACTION

ACTION KRC4:
fbP2KRC4(
	sName:= 'Kuka KRC4 robot vezérlő', 
	bEn:= i_bDoorOK, 
	bZoneEnable:= fbP1AxisX.Axis.NcToPlc.ActPos <= 390,
	timBaseState:= T#20S, 
	bAck:= bAckP);
END_ACTION

ACTION MES:
fbP2MesInterface(
	HOST:= '127.0.0.1', 
	PORT:= 5500, 
	ENABLE:= TRUE, 
	RESET:= fbP2MesInterface.ERROR, 
	STX:= , 
	ETX:= , 
	RESP:= stP2MesResp, 
	TEST_ADAPTER:= '0', 
	ADAPTER_ID:= '1', 
	BUSY=> , 
	READY=> , 
	DONE=> , 
	ERROR=> , 
	ERROR_ID=> );
END_ACTION

ACTION Pneu:
fbP2Lift(
	sName:= 'Z4.5', 
	sBasePosSensor:= 'S4231', 
	sWorkPosSensor:= 'S4232', 
	bEn:= i_bDoorOK, 
	bEHA:= bGlobalEHA, 
	bDisableManualCmd:= NOT bManualMode, 
	bAck:= bAckP, 
	timBasePos:= , 
	timWorkPos:= , 
	stBasePosEvent:= TC_Events.MyEvent.fbP2LiftBPE,
	stWorkPosEvent:= TC_EVENTS.MyEvent.fbP2LiftWPE);
END_ACTION

ACTION RFID:
fbP2RFID(sName:= 'P2 RFID');
END_ACTION

END_PROGRAM

// ---- POUs/Diag.TcPOU
PROGRAM Diag
VAR
		{attribute 'TcLinkTo' := '.wFrmXWcState := TIIF(4)^Inputs^Frm1WcState;
							  .nEcMasterSlaveCountCfg := TIIF(4)^InfoData^CfgSlaveCount;
							  .arrEcMasterNetId := TIIF(4)^InfoData^AmsNetId;
							  .nEcMasterDeviceId := TIIF(4)^InfoData^DevId;
							  .nEcMasterDevState := TIIF(4)^Inputs^DevState;
							  .nEcMasterSlaveCount := TIIF(4)^Inputs^SlaveCount'} 					
	FB_ECAT_DIAG			:FB_EtherCATDiagnosticWrapper;	
	eSubSystem				:E_SubSystem:= E_SubSystem.LOGIC;
	FB_LOGGER_INIT			:FB_EventLogger:= (eSubsystem:= eSubsystem, sJson:='{}');
	FB_EVENTHANDLER			:FB_EventHandler;
	EVENT_TEXT				:STRING(255);
	EVENT_SOURCE			:STRING(255);
END_VAR

